SPLINE
SPL {X  -165.650, Y  +484.445, Z    +0.000, E1   +32.277, E3 +451169.154}
SPL {X  -165.650, Y  +481.524, Z    +0.000, E1   +31.089, E3 +451186.605}
SPL {X  -165.650, Y  +478.014, Z    +0.000, E1   +30.826, E3 +451200.213}
SPL {X  -165.650, Y  +474.473, Z    +0.000, E1   +30.943, E3 +451211.537}
SPL {X  -165.650, Y  +470.376, Z    +0.000, E1   +30.888, E3 +451226.066}
SPL {X  -165.650, Y  +465.146, Z    +0.000, E1   +30.883, E3 +451243.997}
SPL {X  -165.650, Y  +461.106, Z    +0.000, E1   +30.916, E3 +451257.415}
SPL {X  -165.650, Y  +458.435, Z    +0.000, E1   +30.759, E3 +451267.623}
SPL {X  -165.650, Y  +454.220, Z    +0.000, E1   +30.954, E3 +451280.856}
SPL {X  -165.650, Y  +450.433, Z    +0.000, E1   +30.789, E3 +451294.821}
SPL {X  -165.650, Y  +447.097, Z    +0.000, E1   +30.843, E3 +451305.869}
SPL {X  -165.650, Y  +443.673, Z    +0.000, E1   +30.907, E3 +451317.177}
SPL {X  -165.650, Y  +440.976, Z    +0.000, E1   +30.719, E3 +451327.633}
SPL {X  -165.650, Y  +436.324, Z    +0.000, E1   +30.994, E3 +451341.920}
SPL {X  -165.650, Y  +432.765, Z    +0.000, E1   +30.831, E3 +451354.920}
SPL {X  -165.650, Y  +429.309, Z    +0.000, E1   +30.920, E3 +451366.261}
SPL {X  -165.650, Y  +424.918, Z    +0.000, E1   +30.862, E3 +451381.718}
SPL {X  -165.650, Y  +421.437, Z    +0.000, E1   +30.833, E3 +451393.686}
SPL {X  -165.650, Y  +418.489, Z    +0.000, E1   +30.835, E3 +451403.803}
SPL {X  -165.650, Y  +415.831, Z    +0.000, E1   +30.847, E3 +451412.765}
SPL {X  -165.650, Y  +412.139, Z    +0.000, E1   +30.870, E3 +451425.476}
SPL {X  -165.650, Y  +406.834, Z    +0.000, E1   +30.919, E3 +451443.305}
SPL {X  -165.650, Y  +402.516, Z    +0.000, E1   +30.874, E3 +451458.227}
SPL {X  -165.650, Y  +398.147, Z    +0.000, E1   +30.902, E3 +451473.105}
SPL {X  -165.650, Y  +394.694, Z    +0.000, E1   +30.805, E3 +451485.414}
SPL {X  -165.650, Y  +391.522, Z    +0.000, E1   +30.837, E3 +451496.095}
SPL {X  -165.650, Y  +387.533, Z    +0.000, E1   +30.858, E3 +451509.721}
SPL {X  -165.650, Y  +383.627, Z    +0.000, E1   +30.885, E3 +451522.781}
SPL {X  -165.650, Y  +380.752, Z    +0.000, E1   +30.927, E3 +451532.295}
SPL {X  -165.648, Y  +377.739, Z    +0.000, E1   +30.835, E3 +451543.304}
SPL {X  -165.594, Y  +374.183, Z    +0.000, E1   +30.878, E3 +451555.141}
SPL {X  -165.492, Y  +371.263, Z    +0.000, E1   +30.913, E3 +451564.836}
SPL {X  -165.379, Y  +369.027, Z    +0.000, E1   +30.727, E3 +451573.775}
SPL {X  -165.167, Y  +365.866, Z    +0.000, E1   +30.741, E3 +451584.549}
SPL {X  -164.892, Y  +362.671, Z    +0.000, E1   +30.830, E3 +451594.873}
SPL {X  -164.570, Y  +359.612, Z    +0.000, E1   +30.773, E3 +451605.686}
SPL {X  -164.104, Y  +355.923, Z    +0.000, E1   +30.626, E3 +451619.402}
SPL {X  -163.573, Y  +352.353, Z    +0.000, E1   +30.451, E3 +451632.667}
SPL {X  -162.976, Y  +348.856, Z    +0.000, E1   +30.757, E3 +451642.591}
SPL {X  -161.497, Y  +341.640, Z    +0.000, E1   +33.276, E3 +451649.868}
SPL {X  -152.976, Y  +314.952, Z    +0.000, E1   +38.607, E3 +451694.213}
SPL {X  -137.967, Y  +286.821, Z    +0.000, E1   +43.969, E3 +451737.434}
ENDSPLINE

SPLINE
SPL {X  -153.316, Y  +315.777, Z    +0.000, E1   +33.140, E3 +451780.061}
SPL {X  -164.446, Y  +358.564, Z    +0.000, E1   +15.149, E3 +451745.272}
SPL {X  -165.510, Y  +371.680, Z    +0.000, E1    +7.684, E3 +451749.328}
SPL {X  -165.628, Y  +375.818, Z    +0.000, E1    +5.016, E3 +451757.257}
SPL {X  -165.650, Y  +383.362, Z    +0.000, E1    +0.177, E3 +451738.291}
SPL {X  -165.650, Y  +383.923, Z    +0.000, E1    -0.215, E3 +451751.448}
SPL {X  -165.650, Y  +388.083, Z    +0.000, E1    -3.355, E3 +451750.312}
SPL {X  -165.650, Y  +393.983, Z    +0.000, E1    -8.501, E3 +451746.710}
SPL {X  -165.650, Y  +402.241, Z    +0.000, E1   -16.711, E3 +451741.222}
SPL {X  -165.650, Y  +414.811, Z    +0.000, E1   -28.314, E3 +451740.752}
SPL {X  -165.650, Y  +423.479, Z    +0.000, E1   -29.012, E3 +451764.681}
SPL {X  -165.650, Y  +441.276, Z    +0.000, E1   -37.343, E3 +451776.370}
SPL {X  -165.650, Y  +462.890, Z    +0.000, E1   -40.484, E3 +451810.453}
ENDSPLINE

SPLINE
SPL {X  -165.650, Y  +446.920, Z    +0.000, E1   -31.238, E3 +451822.779}
ENDSPLINE

SPLINE
SPL {X  -165.650, Y  +447.935, Z    +0.000, E1   -30.213, E3 +451833.067}
SPL {X  -165.650, Y  +451.020, Z    +0.000, E1   -30.224, E3 +451843.887}
SPL {X  -165.650, Y  +454.519, Z    +0.000, E1   -30.374, E3 +451855.069}
SPL {X  -165.650, Y  +457.429, Z    +0.000, E1   -30.029, E3 +451867.771}
SPL {X  -165.650, Y  +461.678, Z    +0.000, E1   -30.426, E3 +451879.896}
SPL {X  -165.650, Y  +463.853, Z    +0.000, E1   -30.103, E3 +451889.735}
SPL {X  -165.650, Y  +468.397, Z    +0.000, E1   -30.302, E3 +451904.539}
SPL {X  -165.650, Y  +472.566, Z    +0.000, E1   -30.124, E3 +451920.248}
SPL {X  -165.650, Y  +476.540, Z    +0.000, E1   -30.193, E3 +451933.792}
SPL {X  -165.650, Y  +481.042, Z    +0.000, E1   -30.192, E3 +451949.738}
SPL {X  -165.650, Y  +485.236, Z    +0.000, E1   -30.294, E3 +451963.593}
SPL {X  -165.650, Y  +489.057, Z    +0.000, E1   -30.341, E3 +451976.799}
SPL {X  -165.650, Y  +491.647, Z    +0.000, E1   -29.894, E3 +451988.733}
SPL {X  -165.650, Y  +495.051, Z    +0.000, E1   -30.213, E3 +451998.661}
SPL {X  -165.650, Y  +498.418, Z    +0.000, E1   -30.282, E3 +452009.954}
SPL {X  -165.650, Y  +502.421, Z    +0.000, E1   -30.263, E3 +452024.312}
SPL {X  -165.650, Y  +506.344, Z    +0.000, E1   -30.129, E3 +452038.841}
SPL {X  -165.650, Y  +509.866, Z    +0.000, E1   -30.236, E3 +452050.511}
SPL {X  -165.650, Y  +513.685, Z    +0.000, E1   -30.234, E3 +452064.007}
SPL {X  -165.650, Y  +517.104, Z    +0.000, E1   -30.280, E3 +452075.559}
SPL {X  -165.650, Y  +520.621, Z    +0.000, E1   -30.198, E3 +452088.638}
SPL {X  -165.650, Y  +525.344, Z    +0.000, E1   -30.269, E3 +452104.695}
SPL {X  -165.650, Y  +528.152, Z    +0.000, E1   -29.991, E3 +452116.336}
SPL {X  -165.650, Y  +531.783, Z    +0.000, E1   -30.416, E3 +452126.229}
SPL {X  -165.650, Y  +534.115, Z    +0.000, E1   -30.089, E3 +452136.611}
SPL {X  -165.650, Y  +537.522, Z    +0.000, E1   -30.251, E3 +452147.525}
SPL {X  -165.650, Y  +540.621, Z    +0.000, E1   -30.014, E3 +452160.086}
SPL {X  -165.650, Y  +544.944, Z    +0.000, E1   -30.447, E3 +452172.286}
SPL {X  -165.650, Y  +547.199, Z    +0.000, E1   -30.132, E3 +452182.259}
SPL {X  -165.650, Y  +550.512, Z    +0.000, E1   -30.197, E3 +452193.585}
SPL {X  -165.650, Y  +553.852, Z    +0.000, E1   -30.156, E3 +452205.526}
SPL {X  -165.650, Y  +557.277, Z    +0.000, E1   -30.150, E3 +452217.700}
SPL {X  -165.650, Y  +561.168, Z    +0.000, E1   -30.194, E3 +452231.082}
SPL {X  -165.650, Y  +565.528, Z    +0.000, E1   -30.192, E3 +452246.564}
SPL {X  -165.650, Y  +570.048, Z    +0.000, E1   -30.238, E3 +452261.996}
SPL {X  -165.650, Y  +573.110, Z    +0.000, E1   -30.057, E3 +452273.981}
SPL {X  -165.650, Y  +577.587, Z    +0.000, E1   -30.270, E3 +452288.419}
SPL {X  -165.650, Y  +581.190, Z    +0.000, E1   -30.107, E3 +452302.059}
SPL {X  -165.650, Y  +585.053, Z    +0.000, E1   -30.090, E3 +452315.929}
ENDSPLINE

SPLINE
SPL {X  -165.650, Y  +484.445, Z    +0.000, E1   +32.277, E3 +452333.334}
SPL {X  -165.650, Y  +481.524, Z    +0.000, E1   +31.089, E3 +452350.784}
SPL {X  -165.650, Y  +478.014, Z    +0.000, E1   +30.826, E3 +452364.392}
SPL {X  -165.650, Y  +474.473, Z    +0.000, E1   +30.943, E3 +452375.716}
SPL {X  -165.650, Y  +470.376, Z    +0.000, E1   +30.888, E3 +452390.246}
SPL {X  -165.650, Y  +465.146, Z    +0.000, E1   +30.883, E3 +452408.176}
SPL {X  -165.650, Y  +461.106, Z    +0.000, E1   +30.916, E3 +452421.594}
SPL {X  -165.650, Y  +458.435, Z    +0.000, E1   +30.759, E3 +452431.802}
SPL {X  -165.650, Y  +454.220, Z    +0.000, E1   +30.954, E3 +452445.035}
SPL {X  -165.650, Y  +450.433, Z    +0.000, E1   +30.789, E3 +452459.000}
SPL {X  -165.650, Y  +447.097, Z    +0.000, E1   +30.843, E3 +452470.048}
SPL {X  -165.650, Y  +443.673, Z    +0.000, E1   +30.907, E3 +452481.356}
SPL {X  -165.650, Y  +440.976, Z    +0.000, E1   +30.719, E3 +452491.812}
SPL {X  -165.650, Y  +436.324, Z    +0.000, E1   +30.994, E3 +452506.099}
SPL {X  -165.650, Y  +432.765, Z    +0.000, E1   +30.831, E3 +452519.099}
SPL {X  -165.650, Y  +429.309, Z    +0.000, E1   +30.920, E3 +452530.440}
SPL {X  -165.650, Y  +424.918, Z    +0.000, E1   +30.862, E3 +452545.897}
SPL {X  -165.650, Y  +421.437, Z    +0.000, E1   +30.833, E3 +452557.865}
SPL {X  -165.650, Y  +417.366, Z    +0.000, E1   +30.879, E3 +452571.706}
SPL {X  -165.650, Y  +412.139, Z    +0.000, E1   +30.870, E3 +452589.655}
SPL {X  -165.650, Y  +406.834, Z    +0.000, E1   +30.919, E3 +452607.484}
SPL {X  -165.650, Y  +402.516, Z    +0.000, E1   +30.874, E3 +452622.406}
SPL {X  -165.650, Y  +398.147, Z    +0.000, E1   +30.902, E3 +452637.285}
SPL {X  -165.650, Y  +394.694, Z    +0.000, E1   +30.805, E3 +452649.593}
SPL {X  -165.650, Y  +391.522, Z    +0.000, E1   +30.837, E3 +452660.274}
SPL {X  -165.650, Y  +387.533, Z    +0.000, E1   +30.858, E3 +452673.900}
SPL {X  -165.650, Y  +383.627, Z    +0.000, E1   +30.885, E3 +452686.960}
SPL {X  -165.650, Y  +380.752, Z    +0.000, E1   +30.927, E3 +452696.474}
SPL {X  -165.648, Y  +377.739, Z    +0.000, E1   +30.835, E3 +452707.484}
SPL {X  -165.594, Y  +374.183, Z    +0.000, E1   +30.878, E3 +452719.320}
SPL {X  -165.492, Y  +371.263, Z    +0.000, E1   +30.913, E3 +452729.015}
SPL {X  -165.379, Y  +369.027, Z    +0.000, E1   +30.727, E3 +452737.954}
SPL {X  -165.167, Y  +365.866, Z    +0.000, E1   +30.741, E3 +452748.728}
SPL {X  -164.892, Y  +362.671, Z    +0.000, E1   +30.830, E3 +452759.052}
SPL {X  -164.570, Y  +359.612, Z    +0.000, E1   +30.773, E3 +452769.865}
SPL {X  -164.104, Y  +355.923, Z    +0.000, E1   +30.626, E3 +452783.581}
SPL {X  -163.573, Y  +352.353, Z    +0.000, E1   +30.451, E3 +452796.846}
SPL {X  -162.976, Y  +348.856, Z    +0.000, E1   +30.757, E3 +452806.770}
SPL {X  -161.497, Y  +341.640, Z    +0.000, E1   +33.276, E3 +452814.047}
SPL {X  -152.976, Y  +314.952, Z    +0.000, E1   +38.607, E3 +452858.392}
SPL {X  -137.967, Y  +286.821, Z    +0.000, E1   +43.969, E3 +452901.613}
ENDSPLINE

SPLINE
SPL {X  -149.143, Y  +306.414, Z    +0.000, E1   +36.361, E3 +452952.745}
SPL {X  -164.268, Y  +357.145, Z    +0.000, E1   +15.880, E3 +452910.505}
SPL {X  -165.510, Y  +371.680, Z    +0.000, E1    +7.684, E3 +452913.507}
SPL {X  -165.628, Y  +375.818, Z    +0.000, E1    +5.016, E3 +452921.436}
SPL {X  -165.650, Y  +383.362, Z    +0.000, E1    +0.177, E3 +452902.470}
SPL {X  -165.650, Y  +383.923, Z    +0.000, E1    -0.215, E3 +452915.627}
SPL {X  -165.650, Y  +388.083, Z    +0.000, E1    -3.355, E3 +452914.491}
SPL {X  -165.650, Y  +395.510, Z    +0.000, E1    -9.810, E3 +452910.617}
SPL {X  -165.650, Y  +403.066, Z    +0.000, E1   -17.886, E3 +452903.450}
SPL {X  -165.650, Y  +416.345, Z    +0.000, E1   -29.511, E3 +452905.193}
SPL {X  -165.650, Y  +422.331, Z    +0.000, E1   -27.760, E3 +452930.692}
SPL {X  -165.650, Y  +441.276, Z    +0.000, E1   -37.343, E3 +452940.549}
SPL {X  -165.650, Y  +462.890, Z    +0.000, E1   -40.484, E3 +452974.632}
ENDSPLINE

SPLINE
SPL {X  -165.650, Y  +446.920, Z    +0.000, E1   -31.238, E3 +452986.958}
ENDSPLINE

SPLINE
SPL {X  -165.650, Y  +447.935, Z    +0.000, E1   -30.213, E3 +452997.246}
SPL {X  -165.650, Y  +451.020, Z    +0.000, E1   -30.224, E3 +453008.066}
SPL {X  -165.650, Y  +454.519, Z    +0.000, E1   -30.374, E3 +453019.248}
SPL {X  -165.650, Y  +457.429, Z    +0.000, E1   -30.029, E3 +453031.950}
SPL {X  -165.650, Y  +461.678, Z    +0.000, E1   -30.426, E3 +453044.075}
SPL {X  -165.650, Y  +463.853, Z    +0.000, E1   -30.103, E3 +453053.914}
SPL {X  -165.650, Y  +468.397, Z    +0.000, E1   -30.302, E3 +453068.718}
SPL {X  -165.650, Y  +472.566, Z    +0.000, E1   -30.124, E3 +453084.428}
SPL {X  -165.650, Y  +476.540, Z    +0.000, E1   -30.193, E3 +453097.972}
SPL {X  -165.650, Y  +481.042, Z    +0.000, E1   -30.192, E3 +453113.917}
SPL {X  -165.650, Y  +485.236, Z    +0.000, E1   -30.294, E3 +453127.772}
SPL {X  -165.650, Y  +489.057, Z    +0.000, E1   -30.341, E3 +453140.978}
SPL {X  -165.650, Y  +491.647, Z    +0.000, E1   -29.894, E3 +453152.912}
SPL {X  -165.650, Y  +495.051, Z    +0.000, E1   -30.213, E3 +453162.841}
SPL {X  -165.650, Y  +499.546, Z    +0.000, E1   -30.283, E3 +453178.283}
SPL {X  -165.650, Y  +503.544, Z    +0.000, E1   -30.247, E3 +453192.352}
SPL {X  -165.650, Y  +506.344, Z    +0.000, E1   -30.129, E3 +453203.020}
SPL {X  -165.650, Y  +510.660, Z    +0.000, E1   -30.223, E3 +453217.724}
SPL {X  -165.650, Y  +514.670, Z    +0.000, E1   -30.278, E3 +453231.234}
SPL {X  -165.650, Y  +517.919, Z    +0.000, E1   -30.227, E3 +453243.093}
SPL {X  -165.650, Y  +522.822, Z    +0.000, E1   -30.289, E3 +453259.982}
SPL {X  -165.650, Y  +527.393, Z    +0.000, E1   -30.104, E3 +453277.230}
SPL {X  -165.650, Y  +531.783, Z    +0.000, E1   -30.416, E3 +453290.408}
SPL {X  -165.650, Y  +534.115, Z    +0.000, E1   -30.089, E3 +453300.790}
SPL {X  -165.650, Y  +537.522, Z    +0.000, E1   -30.251, E3 +453311.704}
SPL {X  -165.650, Y  +540.621, Z    +0.000, E1   -30.014, E3 +453324.265}
SPL {X  -165.650, Y  +544.944, Z    +0.000, E1   -30.447, E3 +453336.465}
SPL {X  -165.650, Y  +547.199, Z    +0.000, E1   -30.132, E3 +453346.438}
SPL {X  -165.650, Y  +550.512, Z    +0.000, E1   -30.197, E3 +453357.764}
SPL {X  -165.650, Y  +553.852, Z    +0.000, E1   -30.156, E3 +453369.705}
SPL {X  -165.650, Y  +557.277, Z    +0.000, E1   -30.150, E3 +453381.879}
SPL {X  -165.650, Y  +561.168, Z    +0.000, E1   -30.194, E3 +453395.261}
SPL {X  -165.650, Y  +564.449, Z    +0.000, E1   -30.167, E3 +453406.944}
SPL {X  -165.650, Y  +566.935, Z    +0.000, E1   -30.135, E3 +453415.850}
SPL {X  -165.650, Y  +570.048, Z    +0.000, E1   -30.238, E3 +453426.175}
SPL {X  -165.650, Y  +573.110, Z    +0.000, E1   -30.057, E3 +453438.160}
SPL {X  -165.650, Y  +576.497, Z    +0.000, E1   -30.234, E3 +453448.857}
SPL {X  -165.650, Y  +580.354, Z    +0.000, E1   -30.196, E3 +453462.873}
SPL {X  -165.650, Y  +585.053, Z    +0.000, E1   -30.090, E3 +453480.108}
ENDSPLINE

SPLINE
SPL {X  -165.650, Y  +484.445, Z    +0.000, E1   +32.277, E3 +453497.513}
SPL {X  -165.650, Y  +481.524, Z    +0.000, E1   +31.089, E3 +453514.963}
SPL {X  -165.650, Y  +478.014, Z    +0.000, E1   +30.826, E3 +453528.571}
SPL {X  -165.650, Y  +474.473, Z    +0.000, E1   +30.943, E3 +453539.895}
SPL {X  -165.650, Y  +471.826, Z    +0.000, E1   +30.770, E3 +453550.079}
SPL {X  -165.650, Y  +467.753, Z    +0.000, E1   +30.878, E3 +453563.452}
SPL {X  -165.650, Y  +463.837, Z    +0.000, E1   +30.924, E3 +453576.386}
SPL {X  -165.650, Y  +461.106, Z    +0.000, E1   +30.916, E3 +453585.773}
SPL {X  -165.650, Y  +458.435, Z    +0.000, E1   +30.759, E3 +453595.981}
SPL {X  -165.650, Y  +454.220, Z    +0.000, E1   +30.954, E3 +453609.214}
SPL {X  -165.650, Y  +450.433, Z    +0.000, E1   +30.789, E3 +453623.179}
SPL {X  -165.650, Y  +447.097, Z    +0.000, E1   +30.843, E3 +453634.227}
SPL {X  -165.650, Y  +443.673, Z    +0.000, E1   +30.907, E3 +453645.535}
SPL {X  -165.650, Y  +440.976, Z    +0.000, E1   +30.719, E3 +453655.992}
SPL {X  -165.650, Y  +436.324, Z    +0.000, E1   +30.994, E3 +453670.278}
SPL {X  -165.650, Y  +432.765, Z    +0.000, E1   +30.831, E3 +453683.278}
SPL {X  -165.650, Y  +429.309, Z    +0.000, E1   +30.920, E3 +453694.619}
SPL {X  -165.650, Y  +424.918, Z    +0.000, E1   +30.862, E3 +453710.076}
SPL {X  -165.650, Y  +421.437, Z    +0.000, E1   +30.833, E3 +453722.044}
SPL {X  -165.650, Y  +418.489, Z    +0.000, E1   +30.835, E3 +453732.161}
SPL {X  -165.650, Y  +414.127, Z    +0.000, E1   +30.869, E3 +453747.070}
SPL {X  -165.650, Y  +408.547, Z    +0.000, E1   +30.964, E3 +453765.485}
SPL {X  -165.650, Y  +405.433, Z    +0.000, E1   +30.730, E3 +453777.462}
SPL {X  -165.650, Y  +401.473, Z    +0.000, E1   +30.933, E3 +453789.911}
SPL {X  -165.650, Y  +396.018, Z    +0.000, E1   +30.861, E3 +453809.096}
SPL {X  -165.650, Y  +391.522, Z    +0.000, E1   +30.837, E3 +453824.453}
SPL {X  -165.650, Y  +387.533, Z    +0.000, E1   +30.858, E3 +453838.079}
SPL {X  -165.650, Y  +383.627, Z    +0.000, E1   +30.885, E3 +453851.139}
SPL {X  -165.650, Y  +380.752, Z    +0.000, E1   +30.927, E3 +453860.653}
SPL {X  -165.648, Y  +377.739, Z    +0.000, E1   +30.835, E3 +453871.663}
SPL {X  -165.594, Y  +374.183, Z    +0.000, E1   +30.878, E3 +453883.499}
SPL {X  -165.429, Y  +369.945, Z    +0.000, E1   +30.850, E3 +453898.375}
SPL {X  -165.167, Y  +365.866, Z    +0.000, E1   +30.741, E3 +453912.907}
SPL {X  -164.892, Y  +362.671, Z    +0.000, E1   +30.830, E3 +453923.231}
SPL {X  -164.570, Y  +359.612, Z    +0.000, E1   +30.773, E3 +453934.044}
SPL {X  -164.104, Y  +355.923, Z    +0.000, E1   +30.626, E3 +453947.760}
SPL {X  -163.573, Y  +352.353, Z    +0.000, E1   +30.451, E3 +453961.025}
SPL {X  -162.976, Y  +348.856, Z    +0.000, E1   +30.757, E3 +453970.949}
SPL {X  -161.497, Y  +341.640, Z    +0.000, E1   +33.276, E3 +453978.226}
SPL {X  -152.976, Y  +314.952, Z    +0.000, E1   +38.607, E3 +454022.571}
SPL {X  -137.967, Y  +286.821, Z    +0.000, E1   +43.969, E3 +454065.792}
ENDSPLINE

SPLINE
SPL {X  -149.143, Y  +306.414, Z    +0.000, E1   +36.361, E3 +454116.925}
SPL {X  -164.268, Y  +357.145, Z    +0.000, E1   +15.880, E3 +454074.684}
SPL {X  -165.510, Y  +371.680, Z    +0.000, E1    +7.684, E3 +454077.686}
SPL {X  -165.628, Y  +375.818, Z    +0.000, E1    +5.016, E3 +454085.615}
SPL {X  -165.650, Y  +383.362, Z    +0.000, E1    +0.177, E3 +454066.649}
SPL {X  -165.650, Y  +383.923, Z    +0.000, E1    -0.215, E3 +454079.807}
SPL {X  -165.650, Y  +388.083, Z    +0.000, E1    -3.355, E3 +454078.670}
SPL {X  -165.650, Y  +395.510, Z    +0.000, E1    -9.810, E3 +454074.796}
SPL {X  -165.650, Y  +403.066, Z    +0.000, E1   -17.886, E3 +454067.629}
SPL {X  -165.650, Y  +416.345, Z    +0.000, E1   -29.511, E3 +454069.372}
SPL {X  -165.650, Y  +422.331, Z    +0.000, E1   -27.760, E3 +454094.871}
SPL {X  -165.650, Y  +441.276, Z    +0.000, E1   -37.343, E3 +454104.728}
SPL {X  -165.650, Y  +462.890, Z    +0.000, E1   -40.484, E3 +454138.811}
ENDSPLINE

SPLINE
SPL {X  -165.650, Y  +446.920, Z    +0.000, E1   -31.238, E3 +454151.137}
ENDSPLINE

SPLINE
SPL {X  -165.650, Y  +447.935, Z    +0.000, E1   -30.213, E3 +454161.425}
SPL {X  -165.650, Y  +451.020, Z    +0.000, E1   -30.224, E3 +454172.245}
SPL {X  -165.650, Y  +454.519, Z    +0.000, E1   -30.374, E3 +454183.427}
SPL {X  -165.650, Y  +457.429, Z    +0.000, E1   -30.029, E3 +454196.129}
SPL {X  -165.650, Y  +461.678, Z    +0.000, E1   -30.426, E3 +454208.254}
SPL {X  -165.650, Y  +463.853, Z    +0.000, E1   -30.103, E3 +454218.093}
SPL {X  -165.650, Y  +468.397, Z    +0.000, E1   -30.302, E3 +454232.897}
SPL {X  -165.650, Y  +472.566, Z    +0.000, E1   -30.124, E3 +454248.607}
SPL {X  -165.650, Y  +475.265, Z    +0.000, E1   -30.034, E3 +454258.644}
SPL {X  -165.650, Y  +477.862, Z    +0.000, E1   -30.319, E3 +454265.836}
SPL {X  -165.650, Y  +481.042, Z    +0.000, E1   -30.192, E3 +454278.096}
SPL {X  -165.650, Y  +485.236, Z    +0.000, E1   -30.294, E3 +454291.951}
SPL {X  -165.650, Y  +488.041, Z    +0.000, E1   -30.253, E3 +454302.073}
SPL {X  -165.650, Y  +491.281, Z    +0.000, E1   -30.148, E3 +454314.211}
SPL {X  -165.650, Y  +495.051, Z    +0.000, E1   -30.213, E3 +454327.020}
SPL {X  -165.650, Y  +499.546, Z    +0.000, E1   -30.283, E3 +454342.462}
SPL {X  -165.650, Y  +503.544, Z    +0.000, E1   -30.247, E3 +454356.531}
SPL {X  -165.650, Y  +506.344, Z    +0.000, E1   -30.129, E3 +454367.200}
SPL {X  -165.650, Y  +510.660, Z    +0.000, E1   -30.223, E3 +454381.903}
SPL {X  -165.650, Y  +514.670, Z    +0.000, E1   -30.278, E3 +454395.413}
SPL {X  -165.650, Y  +517.919, Z    +0.000, E1   -30.227, E3 +454407.272}
SPL {X  -165.650, Y  +522.822, Z    +0.000, E1   -30.289, E3 +454424.161}
SPL {X  -165.650, Y  +527.393, Z    +0.000, E1   -30.104, E3 +454441.410}
SPL {X  -165.650, Y  +531.783, Z    +0.000, E1   -30.416, E3 +454454.587}
SPL {X  -165.650, Y  +534.115, Z    +0.000, E1   -30.089, E3 +454464.969}
SPL {X  -165.650, Y  +537.522, Z    +0.000, E1   -30.251, E3 +454475.883}
SPL {X  -165.650, Y  +540.621, Z    +0.000, E1   -30.014, E3 +454488.444}
SPL {X  -165.650, Y  +544.944, Z    +0.000, E1   -30.447, E3 +454500.644}
SPL {X  -165.650, Y  +547.199, Z    +0.000, E1   -30.132, E3 +454510.617}
SPL {X  -165.650, Y  +550.512, Z    +0.000, E1   -30.197, E3 +454521.943}
SPL {X  -165.650, Y  +553.852, Z    +0.000, E1   -30.156, E3 +454533.884}
SPL {X  -165.650, Y  +557.277, Z    +0.000, E1   -30.150, E3 +454546.058}
SPL {X  -165.650, Y  +561.168, Z    +0.000, E1   -30.194, E3 +454559.440}
SPL {X  -165.650, Y  +565.528, Z    +0.000, E1   -30.192, E3 +454574.923}
SPL {X  -165.650, Y  +570.048, Z    +0.000, E1   -30.238, E3 +454590.354}
SPL {X  -165.650, Y  +573.110, Z    +0.000, E1   -30.057, E3 +454602.339}
SPL {X  -165.650, Y  +577.587, Z    +0.000, E1   -30.270, E3 +454616.778}
SPL {X  -165.650, Y  +581.190, Z    +0.000, E1   -30.107, E3 +454630.417}
SPL {X  -165.650, Y  +585.053, Z    +0.000, E1   -30.090, E3 +454644.287}
ENDSPLINE

SPLINE
SPL {X  -165.650, Y  +484.445, Z    +0.000, E1   +32.277, E3 +454661.692}
SPL {X  -165.650, Y  +481.524, Z    +0.000, E1   +31.089, E3 +454679.142}
SPL {X  -165.650, Y  +478.014, Z    +0.000, E1   +30.826, E3 +454692.750}
SPL {X  -165.650, Y  +474.473, Z    +0.000, E1   +30.943, E3 +454704.074}
SPL {X  -165.650, Y  +471.826, Z    +0.000, E1   +30.770, E3 +454714.258}
SPL {X  -165.650, Y  +467.753, Z    +0.000, E1   +30.878, E3 +454727.631}
SPL {X  -165.650, Y  +463.837, Z    +0.000, E1   +30.924, E3 +454740.565}
SPL {X  -165.650, Y  +461.106, Z    +0.000, E1   +30.916, E3 +454749.952}
SPL {X  -165.650, Y  +457.156, Z    +0.000, E1   +30.860, E3 +454764.029}
SPL {X  -165.650, Y  +453.156, Z    +0.000, E1   +30.934, E3 +454777.003}
SPL {X  -165.650, Y  +450.433, Z    +0.000, E1   +30.789, E3 +454787.358}
SPL {X  -165.650, Y  +447.097, Z    +0.000, E1   +30.843, E3 +454798.407}
SPL {X  -165.650, Y  +443.673, Z    +0.000, E1   +30.907, E3 +454809.714}
SPL {X  -165.650, Y  +439.486, Z    +0.000, E1   +30.857, E3 +454824.523}
SPL {X  -165.650, Y  +435.146, Z    +0.000, E1   +30.969, E3 +454838.443}
SPL {X  -165.650, Y  +431.607, Z    +0.000, E1   +30.889, E3 +454851.157}
SPL {X  -165.650, Y  +427.340, Z    +0.000, E1   +30.870, E3 +454865.869}
SPL {X  -165.650, Y  +423.901, Z    +0.000, E1   +30.858, E3 +454877.625}
SPL {X  -165.650, Y  +421.437, Z    +0.000, E1   +30.833, E3 +454886.223}
SPL {X  -165.650, Y  +418.489, Z    +0.000, E1   +30.835, E3 +454896.340}
SPL {X  -165.650, Y  +414.127, Z    +0.000, E1   +30.869, E3 +454911.249}
SPL {X  -165.650, Y  +408.547, Z    +0.000, E1   +30.964, E3 +454929.664}
SPL {X  -165.650, Y  +405.433, Z    +0.000, E1   +30.730, E3 +454941.642}
SPL {X  -165.650, Y  +401.473, Z    +0.000, E1   +30.933, E3 +454954.090}
SPL {X  -165.650, Y  +396.018, Z    +0.000, E1   +30.861, E3 +454973.275}
SPL {X  -165.650, Y  +390.331, Z    +0.000, E1   +30.892, E3 +454992.527}
SPL {X  -165.650, Y  +384.849, Z    +0.000, E1   +30.885, E3 +455011.331}
SPL {X  -165.650, Y  +380.752, Z    +0.000, E1   +30.927, E3 +455024.832}
SPL {X  -165.648, Y  +377.739, Z    +0.000, E1   +30.835, E3 +455035.842}
SPL {X  -165.594, Y  +374.183, Z    +0.000, E1   +30.878, E3 +455047.679}
SPL {X  -165.492, Y  +371.263, Z    +0.000, E1   +30.913, E3 +455057.374}
SPL {X  -165.379, Y  +369.027, Z    +0.000, E1   +30.727, E3 +455066.312}
SPL {X  -165.167, Y  +365.866, Z    +0.000, E1   +30.741, E3 +455077.086}
SPL {X  -164.892, Y  +362.671, Z    +0.000, E1   +30.830, E3 +455087.410}
SPL {X  -164.570, Y  +359.612, Z    +0.000, E1   +30.773, E3 +455098.223}
SPL {X  -164.104, Y  +355.923, Z    +0.000, E1   +30.626, E3 +455111.939}
SPL {X  -163.573, Y  +352.353, Z    +0.000, E1   +30.451, E3 +455125.204}
SPL {X  -162.476, Y  +346.230, Z    +0.000, E1   +31.677, E3 +455137.785}
SPL {X  -152.976, Y  +314.952, Z    +0.000, E1   +38.607, E3 +455186.750}
SPL {X  -137.967, Y  +286.821, Z    +0.000, E1   +43.969, E3 +455229.971}
ENDSPLINE

SPLINE
SPL {X  -149.143, Y  +306.414, Z    +0.000, E1   +36.361, E3 +455281.104}
SPL {X  -163.091, Y  +349.496, Z    +0.000, E1   +19.699, E3 +455237.887}
SPL {X  -165.027, Y  +364.142, Z    +0.000, E1   +12.054, E3 +455241.027}
SPL {X  -165.612, Y  +374.969, Z    +0.000, E1    +5.630, E3 +455246.210}
SPL {X  -165.650, Y  +383.362, Z    +0.000, E1    +0.177, E3 +455230.828}
SPL {X  -165.650, Y  +383.923, Z    +0.000, E1    -0.215, E3 +455243.986}
SPL {X  -165.650, Y  +388.083, Z    +0.000, E1    -3.355, E3 +455242.849}
SPL {X  -165.650, Y  +393.983, Z    +0.000, E1    -8.501, E3 +455239.247}
SPL {X  -165.650, Y  +402.241, Z    +0.000, E1   -16.711, E3 +455233.759}
SPL {X  -165.650, Y  +416.345, Z    +0.000, E1   -29.511, E3 +455233.551}
SPL {X  -165.650, Y  +422.331, Z    +0.000, E1   -27.760, E3 +455259.050}
SPL {X  -165.650, Y  +441.276, Z    +0.000, E1   -37.343, E3 +455268.907}
SPL {X  -165.650, Y  +462.890, Z    +0.000, E1   -40.484, E3 +455302.990}
ENDSPLINE

SPLINE
SPL {X  -165.650, Y  +446.920, Z    +0.000, E1   -31.238, E3 +455315.316}
ENDSPLINE

SPLINE
SPL {X  -165.650, Y  +447.935, Z    +0.000, E1   -30.213, E3 +455325.604}
SPL {X  -165.650, Y  +451.020, Z    +0.000, E1   -30.224, E3 +455336.424}
SPL {X  -165.650, Y  +454.519, Z    +0.000, E1   -30.374, E3 +455347.607}
SPL {X  -165.650, Y  +456.542, Z    +0.000, E1   -29.986, E3 +455357.351}
SPL {X  -165.650, Y  +460.618, Z    +0.000, E1   -30.298, E3 +455369.672}
SPL {X  -165.650, Y  +463.853, Z    +0.000, E1   -30.103, E3 +455382.273}
SPL {X  -165.650, Y  +468.397, Z    +0.000, E1   -30.302, E3 +455397.076}
SPL {X  -165.650, Y  +472.566, Z    +0.000, E1   -30.124, E3 +455412.786}
SPL {X  -165.650, Y  +475.265, Z    +0.000, E1   -30.034, E3 +455422.823}
SPL {X  -165.650, Y  +477.862, Z    +0.000, E1   -30.319, E3 +455430.015}
SPL {X  -165.650, Y  +481.042, Z    +0.000, E1   -30.192, E3 +455442.275}
SPL {X  -165.650, Y  +485.236, Z    +0.000, E1   -30.294, E3 +455456.131}
SPL {X  -165.650, Y  +488.041, Z    +0.000, E1   -30.253, E3 +455466.252}
SPL {X  -165.650, Y  +491.281, Z    +0.000, E1   -30.148, E3 +455478.390}
SPL {X  -165.650, Y  +495.051, Z    +0.000, E1   -30.213, E3 +455491.199}
SPL {X  -165.650, Y  +499.546, Z    +0.000, E1   -30.283, E3 +455506.642}
SPL {X  -165.650, Y  +503.544, Z    +0.000, E1   -30.247, E3 +455520.710}
SPL {X  -165.650, Y  +506.344, Z    +0.000, E1   -30.129, E3 +455531.379}
SPL {X  -165.650, Y  +510.660, Z    +0.000, E1   -30.223, E3 +455546.082}
SPL {X  -165.650, Y  +514.670, Z    +0.000, E1   -30.278, E3 +455559.592}
SPL {X  -165.650, Y  +517.919, Z    +0.000, E1   -30.227, E3 +455571.451}
SPL {X  -165.650, Y  +521.521, Z    +0.000, E1   -30.210, E3 +455584.126}
SPL {X  -165.650, Y  +525.344, Z    +0.000, E1   -30.269, E3 +455597.232}
SPL {X  -165.650, Y  +528.152, Z    +0.000, E1   -29.991, E3 +455608.873}
SPL {X  -165.650, Y  +531.783, Z    +0.000, E1   -30.416, E3 +455618.766}
SPL {X  -165.650, Y  +534.115, Z    +0.000, E1   -30.089, E3 +455629.148}
SPL {X  -165.650, Y  +537.522, Z    +0.000, E1   -30.251, E3 +455640.062}
SPL {X  -165.650, Y  +540.621, Z    +0.000, E1   -30.014, E3 +455652.623}
SPL {X  -165.650, Y  +544.944, Z    +0.000, E1   -30.447, E3 +455664.823}
SPL {X  -165.650, Y  +547.199, Z    +0.000, E1   -30.132, E3 +455674.796}
SPL {X  -165.650, Y  +550.512, Z    +0.000, E1   -30.197, E3 +455686.122}
SPL {X  -165.650, Y  +553.852, Z    +0.000, E1   -30.156, E3 +455698.063}
SPL {X  -165.650, Y  +557.277, Z    +0.000, E1   -30.150, E3 +455710.238}
SPL {X  -165.650, Y  +561.168, Z    +0.000, E1   -30.194, E3 +455723.619}
SPL {X  -165.650, Y  +565.528, Z    +0.000, E1   -30.192, E3 +455739.102}
SPL {X  -165.650, Y  +570.048, Z    +0.000, E1   -30.238, E3 +455754.533}
SPL {X  -165.650, Y  +573.110, Z    +0.000, E1   -30.057, E3 +455766.518}
SPL {X  -165.650, Y  +576.497, Z    +0.000, E1   -30.234, E3 +455777.216}
SPL {X  -165.650, Y  +580.354, Z    +0.000, E1   -30.196, E3 +455791.231}
SPL {X  -165.650, Y  +585.053, Z    +0.000, E1   -30.090, E3 +455808.466}
ENDSPLINE

SPLINE
SPL {X  -165.650, Y  +484.968, Z    +0.000, E1   +32.508, E3 +455822.432}
SPL {X  -165.650, Y  +482.280, Z    +0.000, E1   +31.680, E3 +455836.759}
SPL {X  -165.650, Y  +481.693, Z    +0.000, E1   +30.334, E3 +455847.468}
SPL {X  -165.650, Y  +478.014, Z    +0.000, E1   +30.826, E3 +455856.929}
SPL {X  -165.650, Y  +474.473, Z    +0.000, E1   +30.943, E3 +455868.253}
SPL {X  -165.650, Y  +471.826, Z    +0.000, E1   +30.770, E3 +455878.437}
SPL {X  -165.650, Y  +467.753, Z    +0.000, E1   +30.878, E3 +455891.810}
SPL {X  -165.650, Y  +463.837, Z    +0.000, E1   +30.924, E3 +455904.744}
SPL {X  -165.650, Y  +461.106, Z    +0.000, E1   +30.916, E3 +455914.131}
SPL {X  -165.650, Y  +458.435, Z    +0.000, E1   +30.759, E3 +455924.339}
SPL {X  -165.650, Y  +454.220, Z    +0.000, E1   +30.954, E3 +455937.572}
SPL {X  -165.650, Y  +450.433, Z    +0.000, E1   +30.789, E3 +455951.537}
SPL {X  -165.650, Y  +447.097, Z    +0.000, E1   +30.843, E3 +455962.586}
SPL {X  -165.650, Y  +443.673, Z    +0.000, E1   +30.907, E3 +455973.893}
SPL {X  -165.650, Y  +440.976, Z    +0.000, E1   +30.719, E3 +455984.350}
SPL {X  -165.650, Y  +437.973, Z    +0.000, E1   +30.928, E3 +455993.222}
SPL {X  -165.650, Y  +434.043, Z    +0.000, E1   +30.950, E3 +456006.719}
SPL {X  -165.650, Y  +430.419, Z    +0.000, E1   +30.895, E3 +456019.222}
SPL {X  -165.650, Y  +427.340, Z    +0.000, E1   +30.870, E3 +456030.048}
SPL {X  -165.650, Y  +422.641, Z    +0.000, E1   +30.884, E3 +456046.137}
SPL {X  -165.650, Y  +418.489, Z    +0.000, E1   +30.835, E3 +456060.519}
SPL {X  -165.650, Y  +414.127, Z    +0.000, E1   +30.869, E3 +456075.428}
SPL {X  -165.650, Y  +408.547, Z    +0.000, E1   +30.964, E3 +456093.843}
SPL {X  -165.650, Y  +405.433, Z    +0.000, E1   +30.730, E3 +456105.821}
SPL {X  -165.650, Y  +402.516, Z    +0.000, E1   +30.874, E3 +456114.943}
SPL {X  -165.650, Y  +398.147, Z    +0.000, E1   +30.902, E3 +456129.822}
SPL {X  -165.650, Y  +394.694, Z    +0.000, E1   +30.805, E3 +456142.130}
SPL {X  -165.650, Y  +391.522, Z    +0.000, E1   +30.837, E3 +456152.811}
SPL {X  -165.650, Y  +387.533, Z    +0.000, E1   +30.858, E3 +456166.437}
SPL {X  -165.650, Y  +383.627, Z    +0.000, E1   +30.885, E3 +456179.497}
SPL {X  -165.650, Y  +379.886, Z    +0.000, E1   +30.887, E3 +456192.386}
SPL {X  -165.614, Y  +375.058, Z    +0.000, E1   +30.905, E3 +456208.839}
SPL {X  -165.492, Y  +371.263, Z    +0.000, E1   +30.913, E3 +456221.553}
SPL {X  -165.379, Y  +369.027, Z    +0.000, E1   +30.727, E3 +456230.491}
SPL {X  -165.167, Y  +365.866, Z    +0.000, E1   +30.741, E3 +456241.265}
SPL {X  -164.892, Y  +362.671, Z    +0.000, E1   +30.830, E3 +456251.589}
SPL {X  -164.570, Y  +359.612, Z    +0.000, E1   +30.773, E3 +456262.402}
SPL {X  -164.104, Y  +355.923, Z    +0.000, E1   +30.626, E3 +456276.118}
SPL {X  -163.573, Y  +352.353, Z    +0.000, E1   +30.451, E3 +456289.383}
SPL {X  -162.976, Y  +348.856, Z    +0.000, E1   +30.757, E3 +456299.307}
SPL {X  -161.497, Y  +341.640, Z    +0.000, E1   +33.276, E3 +456306.585}
SPL {X  -152.976, Y  +314.952, Z    +0.000, E1   +38.607, E3 +456350.929}
SPL {X  -137.967, Y  +286.821, Z    +0.000, E1   +43.969, E3 +456394.150}
ENDSPLINE

SPLINE
SPL {X  -149.143, Y  +306.414, Z    +0.000, E1   +36.361, E3 +456445.283}
SPL {X  -164.268, Y  +357.145, Z    +0.000, E1   +15.880, E3 +456403.042}
SPL {X  -165.379, Y  +369.025, Z    +0.000, E1    +9.158, E3 +456407.713}
SPL {X  -165.612, Y  +374.969, Z    +0.000, E1    +5.630, E3 +456410.389}
SPL {X  -165.650, Y  +383.362, Z    +0.000, E1    +0.177, E3 +456395.007}
SPL {X  -165.650, Y  +383.923, Z    +0.000, E1    -0.215, E3 +456408.165}
SPL {X  -165.650, Y  +388.083, Z    +0.000, E1    -3.355, E3 +456407.028}
SPL {X  -165.650, Y  +393.983, Z    +0.000, E1    -8.501, E3 +456403.426}
SPL {X  -165.650, Y  +402.241, Z    +0.000, E1   -16.711, E3 +456397.938}
SPL {X  -165.650, Y  +416.345, Z    +0.000, E1   -29.511, E3 +456397.730}
SPL {X  -165.650, Y  +422.331, Z    +0.000, E1   -27.760, E3 +456423.229}
SPL {X  -165.650, Y  +441.276, Z    +0.000, E1   -37.343, E3 +456433.086}
SPL {X  -165.650, Y  +462.890, Z    +0.000, E1   -40.484, E3 +456467.169}
ENDSPLINE

SPLINE
SPL {X  -165.650, Y  +446.920, Z    +0.000, E1   -31.238, E3 +456479.495}
ENDSPLINE

SPLINE
SPL {X  -165.650, Y  +447.935, Z    +0.000, E1   -30.213, E3 +456489.783}
SPL {X  -165.650, Y  +451.020, Z    +0.000, E1   -30.224, E3 +456500.603}
SPL {X  -165.650, Y  +454.519, Z    +0.000, E1   -30.374, E3 +456511.786}
SPL {X  -165.650, Y  +456.542, Z    +0.000, E1   -29.986, E3 +456521.530}
SPL {X  -165.650, Y  +460.618, Z    +0.000, E1   -30.298, E3 +456533.851}
SPL {X  -165.650, Y  +463.853, Z    +0.000, E1   -30.103, E3 +456546.452}
SPL {X  -165.650, Y  +468.397, Z    +0.000, E1   -30.302, E3 +456561.256}
SPL {X  -165.650, Y  +472.566, Z    +0.000, E1   -30.124, E3 +456576.965}
SPL {X  -165.650, Y  +476.540, Z    +0.000, E1   -30.193, E3 +456590.509}
SPL {X  -165.650, Y  +480.320, Z    +0.000, E1   -30.163, E3 +456603.987}
SPL {X  -165.650, Y  +484.477, Z    +0.000, E1   -30.274, E3 +456617.876}
SPL {X  -165.650, Y  +488.041, Z    +0.000, E1   -30.253, E3 +456630.431}
SPL {X  -165.650, Y  +491.281, Z    +0.000, E1   -30.148, E3 +456642.569}
SPL {X  -165.650, Y  +495.051, Z    +0.000, E1   -30.213, E3 +456655.378}
SPL {X  -165.650, Y  +499.546, Z    +0.000, E1   -30.283, E3 +456670.821}
SPL {X  -165.650, Y  +503.544, Z    +0.000, E1   -30.247, E3 +456684.889}
SPL {X  -165.650, Y  +506.344, Z    +0.000, E1   -30.129, E3 +456695.558}
SPL {X  -165.650, Y  +509.866, Z    +0.000, E1   -30.236, E3 +456707.227}
SPL {X  -165.650, Y  +513.685, Z    +0.000, E1   -30.234, E3 +456720.723}
SPL {X  -165.650, Y  +517.919, Z    +0.000, E1   -30.227, E3 +456735.630}
SPL {X  -165.650, Y  +521.521, Z    +0.000, E1   -30.210, E3 +456748.305}
SPL {X  -165.650, Y  +525.344, Z    +0.000, E1   -30.269, E3 +456761.411}
SPL {X  -165.650, Y  +528.152, Z    +0.000, E1   -29.991, E3 +456773.052}
SPL {X  -165.650, Y  +531.783, Z    +0.000, E1   -30.416, E3 +456782.945}
SPL {X  -165.650, Y  +534.115, Z    +0.000, E1   -30.089, E3 +456793.327}
SPL {X  -165.650, Y  +537.522, Z    +0.000, E1   -30.251, E3 +456804.241}
SPL {X  -165.650, Y  +540.621, Z    +0.000, E1   -30.014, E3 +456816.802}
SPL {X  -165.650, Y  +544.944, Z    +0.000, E1   -30.447, E3 +456829.002}
SPL {X  -165.650, Y  +547.199, Z    +0.000, E1   -30.132, E3 +456838.976}
SPL {X  -165.650, Y  +550.512, Z    +0.000, E1   -30.197, E3 +456850.301}
SPL {X  -165.650, Y  +553.852, Z    +0.000, E1   -30.156, E3 +456862.242}
SPL {X  -165.650, Y  +557.277, Z    +0.000, E1   -30.150, E3 +456874.417}
SPL {X  -165.650, Y  +561.168, Z    +0.000, E1   -30.194, E3 +456887.798}
SPL {X  -165.650, Y  +565.528, Z    +0.000, E1   -30.192, E3 +456903.281}
SPL {X  -165.650, Y  +570.048, Z    +0.000, E1   -30.238, E3 +456918.712}
SPL {X  -165.650, Y  +573.110, Z    +0.000, E1   -30.057, E3 +456930.697}
SPL {X  -165.650, Y  +577.587, Z    +0.000, E1   -30.270, E3 +456945.136}
SPL {X  -165.650, Y  +581.190, Z    +0.000, E1   -30.107, E3 +456958.775}
SPL {X  -165.650, Y  +585.053, Z    +0.000, E1   -30.090, E3 +456972.645}
ENDSPLINE

SPLINE
SPL {X  -165.650, Y  +484.445, Z    +0.000, E1   +32.277, E3 +456990.050}
SPL {X  -165.650, Y  +481.524, Z    +0.000, E1   +31.089, E3 +457007.500}
SPL {X  -165.650, Y  +478.014, Z    +0.000, E1   +30.826, E3 +457021.108}
SPL {X  -165.650, Y  +474.473, Z    +0.000, E1   +30.943, E3 +457032.432}
SPL {X  -165.650, Y  +471.826, Z    +0.000, E1   +30.770, E3 +457042.616}
SPL {X  -165.650, Y  +467.753, Z    +0.000, E1   +30.878, E3 +457055.989}
SPL {X  -165.650, Y  +463.837, Z    +0.000, E1   +30.924, E3 +457068.923}
SPL {X  -165.650, Y  +461.106, Z    +0.000, E1   +30.916, E3 +457078.310}
SPL {X  -165.650, Y  +457.156, Z    +0.000, E1   +30.860, E3 +457092.387}
SPL {X  -165.650, Y  +453.156, Z    +0.000, E1   +30.934, E3 +457105.361}
SPL {X  -165.650, Y  +450.433, Z    +0.000, E1   +30.789, E3 +457115.716}
SPL {X  -165.650, Y  +447.097, Z    +0.000, E1   +30.843, E3 +457126.765}
SPL {X  -165.650, Y  +443.673, Z    +0.000, E1   +30.907, E3 +457138.072}
SPL {X  -165.650, Y  +439.486, Z    +0.000, E1   +30.857, E3 +457152.882}
SPL {X  -165.650, Y  +435.146, Z    +0.000, E1   +30.969, E3 +457166.801}
SPL {X  -165.650, Y  +432.765, Z    +0.000, E1   +30.831, E3 +457175.815}
SPL {X  -165.650, Y  +429.309, Z    +0.000, E1   +30.920, E3 +457187.156}
SPL {X  -165.650, Y  +424.918, Z    +0.000, E1   +30.862, E3 +457202.613}
SPL {X  -165.650, Y  +421.437, Z    +0.000, E1   +30.833, E3 +457214.582}
SPL {X  -165.650, Y  +417.366, Z    +0.000, E1   +30.879, E3 +457228.422}
SPL {X  -165.650, Y  +413.181, Z    +0.000, E1   +30.815, E3 +457243.020}
SPL {X  -165.650, Y  +408.547, Z    +0.000, E1   +30.964, E3 +457258.023}
SPL {X  -165.650, Y  +403.421, Z    +0.000, E1   +30.863, E3 +457276.240}
SPL {X  -165.650, Y  +399.681, Z    +0.000, E1   +30.933, E3 +457288.323}
SPL {X  -165.650, Y  +396.018, Z    +0.000, E1   +30.861, E3 +457301.633}
SPL {X  -165.650, Y  +391.522, Z    +0.000, E1   +30.837, E3 +457316.990}
SPL {X  -165.650, Y  +387.533, Z    +0.000, E1   +30.858, E3 +457330.616}
SPL {X  -165.650, Y  +383.627, Z    +0.000, E1   +30.885, E3 +457343.677}
SPL {X  -165.650, Y  +380.752, Z    +0.000, E1   +30.927, E3 +457353.190}
SPL {X  -165.648, Y  +377.739, Z    +0.000, E1   +30.835, E3 +457364.200}
SPL {X  -165.594, Y  +374.183, Z    +0.000, E1   +30.878, E3 +457376.037}
SPL {X  -165.429, Y  +369.945, Z    +0.000, E1   +30.850, E3 +457390.912}
SPL {X  -165.167, Y  +365.866, Z    +0.000, E1   +30.741, E3 +457405.444}
SPL {X  -164.892, Y  +362.671, Z    +0.000, E1   +30.830, E3 +457415.768}
SPL {X  -164.570, Y  +359.612, Z    +0.000, E1   +30.773, E3 +457426.581}
SPL {X  -164.104, Y  +355.923, Z    +0.000, E1   +30.626, E3 +457440.298}
SPL {X  -163.573, Y  +352.353, Z    +0.000, E1   +30.451, E3 +457453.562}
SPL {X  -162.476, Y  +346.230, Z    +0.000, E1   +31.677, E3 +457466.143}
SPL {X  -152.976, Y  +314.952, Z    +0.000, E1   +38.607, E3 +457515.108}
SPL {X  -137.967, Y  +286.821, Z    +0.000, E1   +43.969, E3 +457558.329}
ENDSPLINE

SPLINE
SPL {X  -153.316, Y  +315.777, Z    +0.000, E1   +33.140, E3 +457600.957}
SPL {X  -164.446, Y  +358.564, Z    +0.000, E1   +15.149, E3 +457566.168}
SPL {X  -165.510, Y  +371.680, Z    +0.000, E1    +7.684, E3 +457570.223}
SPL {X  -165.628, Y  +375.818, Z    +0.000, E1    +5.016, E3 +457578.153}
SPL {X  -165.650, Y  +383.362, Z    +0.000, E1    +0.177, E3 +457559.186}
SPL {X  -165.650, Y  +383.923, Z    +0.000, E1    -0.215, E3 +457572.344}
SPL {X  -165.650, Y  +388.083, Z    +0.000, E1    -3.355, E3 +457571.207}
SPL {X  -165.650, Y  +393.983, Z    +0.000, E1    -8.501, E3 +457567.606}
SPL {X  -165.650, Y  +402.241, Z    +0.000, E1   -16.711, E3 +457562.117}
SPL {X  -165.650, Y  +414.811, Z    +0.000, E1   -28.314, E3 +457561.648}
SPL {X  -165.650, Y  +423.479, Z    +0.000, E1   -29.012, E3 +457585.576}
SPL {X  -165.650, Y  +441.276, Z    +0.000, E1   -37.343, E3 +457597.265}
SPL {X  -165.650, Y  +462.890, Z    +0.000, E1   -40.484, E3 +457631.348}
ENDSPLINE

SPLINE
SPL {X  -165.650, Y  +446.920, Z    +0.000, E1   -31.238, E3 +457643.674}
ENDSPLINE

SPLINE
SPL {X  -165.650, Y  +447.935, Z    +0.000, E1   -30.213, E3 +457653.962}
SPL {X  -165.650, Y  +451.020, Z    +0.000, E1   -30.224, E3 +457664.782}
SPL {X  -165.650, Y  +454.519, Z    +0.000, E1   -30.374, E3 +457675.965}
SPL {X  -165.650, Y  +456.542, Z    +0.000, E1   -29.986, E3 +457685.709}
SPL {X  -165.650, Y  +460.618, Z    +0.000, E1   -30.298, E3 +457698.030}
SPL {X  -165.650, Y  +463.853, Z    +0.000, E1   -30.103, E3 +457710.631}
SPL {X  -165.650, Y  +468.397, Z    +0.000, E1   -30.302, E3 +457725.435}
SPL {X  -165.650, Y  +472.566, Z    +0.000, E1   -30.124, E3 +457741.144}
SPL {X  -165.650, Y  +476.540, Z    +0.000, E1   -30.193, E3 +457754.688}
SPL {X  -165.650, Y  +480.320, Z    +0.000, E1   -30.163, E3 +457768.166}
SPL {X  -165.650, Y  +484.477, Z    +0.000, E1   -30.274, E3 +457782.055}
SPL {X  -165.650, Y  +488.041, Z    +0.000, E1   -30.253, E3 +457794.610}
SPL {X  -165.650, Y  +491.281, Z    +0.000, E1   -30.148, E3 +457806.748}
SPL {X  -165.650, Y  +495.051, Z    +0.000, E1   -30.213, E3 +457819.557}
SPL {X  -165.650, Y  +498.418, Z    +0.000, E1   -30.282, E3 +457830.850}
SPL {X  -165.650, Y  +500.833, Z    +0.000, E1   -30.191, E3 +457839.899}
SPL {X  -165.650, Y  +504.246, Z    +0.000, E1   -30.231, E3 +457851.765}
SPL {X  -165.650, Y  +507.017, Z    +0.000, E1   -30.108, E3 +457862.174}
SPL {X  -165.650, Y  +510.660, Z    +0.000, E1   -30.223, E3 +457874.440}
SPL {X  -165.650, Y  +514.670, Z    +0.000, E1   -30.278, E3 +457887.950}
SPL {X  -165.650, Y  +517.919, Z    +0.000, E1   -30.227, E3 +457899.810}
SPL {X  -165.650, Y  +522.822, Z    +0.000, E1   -30.289, E3 +457916.699}
SPL {X  -165.650, Y  +527.393, Z    +0.000, E1   -30.104, E3 +457933.947}
SPL {X  -165.650, Y  +531.783, Z    +0.000, E1   -30.416, E3 +457947.124}
SPL {X  -165.650, Y  +534.115, Z    +0.000, E1   -30.089, E3 +457957.506}
SPL {X  -165.650, Y  +537.522, Z    +0.000, E1   -30.251, E3 +457968.421}
SPL {X  -165.650, Y  +540.621, Z    +0.000, E1   -30.014, E3 +457980.982}
SPL {X  -165.650, Y  +544.944, Z    +0.000, E1   -30.447, E3 +457993.181}
SPL {X  -165.650, Y  +548.549, Z    +0.000, E1   -30.216, E3 +458007.505}
SPL {X  -165.650, Y  +553.092, Z    +0.000, E1   -30.157, E3 +458023.847}
SPL {X  -165.650, Y  +556.274, Z    +0.000, E1   -30.127, E3 +458035.102}
SPL {X  -165.650, Y  +560.243, Z    +0.000, E1   -30.214, E3 +458048.768}
SPL {X  -165.650, Y  +565.528, Z    +0.000, E1   -30.192, E3 +458067.460}
SPL {X  -165.650, Y  +570.048, Z    +0.000, E1   -30.238, E3 +458082.891}
SPL {X  -165.650, Y  +573.110, Z    +0.000, E1   -30.057, E3 +458094.876}
SPL {X  -165.650, Y  +576.497, Z    +0.000, E1   -30.234, E3 +458105.574}
SPL {X  -165.650, Y  +580.354, Z    +0.000, E1   -30.196, E3 +458119.589}
SPL {X  -165.650, Y  +585.053, Z    +0.000, E1   -30.090, E3 +458136.825}
ENDSPLINE

SPLINE
SPL {X  -165.650, Y  +484.445, Z    +0.000, E1   +32.277, E3 +458154.229}
SPL {X  -165.650, Y  +481.524, Z    +0.000, E1   +31.089, E3 +458171.680}
SPL {X  -165.650, Y  +478.014, Z    +0.000, E1   +30.826, E3 +458185.287}
SPL {X  -165.650, Y  +474.473, Z    +0.000, E1   +30.943, E3 +458196.612}
SPL {X  -165.650, Y  +470.376, Z    +0.000, E1   +30.888, E3 +458211.141}
SPL {X  -165.650, Y  +465.146, Z    +0.000, E1   +30.883, E3 +458229.071}
SPL {X  -165.650, Y  +461.106, Z    +0.000, E1   +30.916, E3 +458242.489}
SPL {X  -165.650, Y  +458.435, Z    +0.000, E1   +30.759, E3 +458252.697}
SPL {X  -165.650, Y  +454.220, Z    +0.000, E1   +30.954, E3 +458265.930}
SPL {X  -165.650, Y  +450.433, Z    +0.000, E1   +30.789, E3 +458279.895}
SPL {X  -165.650, Y  +447.097, Z    +0.000, E1   +30.843, E3 +458290.944}
SPL {X  -165.650, Y  +443.673, Z    +0.000, E1   +30.907, E3 +458302.251}
SPL {X  -165.650, Y  +440.976, Z    +0.000, E1   +30.719, E3 +458312.708}
SPL {X  -165.650, Y  +436.324, Z    +0.000, E1   +30.994, E3 +458326.994}
SPL {X  -165.650, Y  +432.765, Z    +0.000, E1   +30.831, E3 +458339.994}
SPL {X  -165.650, Y  +429.309, Z    +0.000, E1   +30.920, E3 +458351.335}
SPL {X  -165.650, Y  +424.918, Z    +0.000, E1   +30.862, E3 +458366.792}
SPL {X  -165.650, Y  +421.437, Z    +0.000, E1   +30.833, E3 +458378.761}
SPL {X  -165.650, Y  +418.489, Z    +0.000, E1   +30.835, E3 +458388.877}
SPL {X  -165.650, Y  +414.127, Z    +0.000, E1   +30.869, E3 +458403.786}
SPL {X  -165.650, Y  +408.547, Z    +0.000, E1   +30.964, E3 +458422.202}
SPL {X  -165.650, Y  +405.433, Z    +0.000, E1   +30.730, E3 +458434.179}
SPL {X  -165.650, Y  +402.516, Z    +0.000, E1   +30.874, E3 +458443.302}
SPL {X  -165.650, Y  +398.147, Z    +0.000, E1   +30.902, E3 +458458.180}
SPL {X  -165.650, Y  +394.694, Z    +0.000, E1   +30.805, E3 +458470.488}
SPL {X  -165.650, Y  +391.522, Z    +0.000, E1   +30.837, E3 +458481.169}
SPL {X  -165.650, Y  +387.533, Z    +0.000, E1   +30.858, E3 +458494.795}
SPL {X  -165.650, Y  +383.627, Z    +0.000, E1   +30.885, E3 +458507.856}
SPL {X  -165.650, Y  +379.886, Z    +0.000, E1   +30.887, E3 +458520.744}
SPL {X  -165.614, Y  +375.058, Z    +0.000, E1   +30.905, E3 +458537.197}
SPL {X  -165.492, Y  +371.263, Z    +0.000, E1   +30.913, E3 +458549.911}
SPL {X  -165.379, Y  +369.027, Z    +0.000, E1   +30.727, E3 +458558.849}
SPL {X  -165.167, Y  +365.866, Z    +0.000, E1   +30.741, E3 +458569.623}
SPL {X  -164.892, Y  +362.671, Z    +0.000, E1   +30.830, E3 +458579.948}
SPL {X  -164.570, Y  +359.612, Z    +0.000, E1   +30.773, E3 +458590.760}
SPL {X  -164.104, Y  +355.923, Z    +0.000, E1   +30.626, E3 +458604.477}
SPL {X  -163.573, Y  +352.353, Z    +0.000, E1   +30.451, E3 +458617.741}
SPL {X  -162.476, Y  +346.230, Z    +0.000, E1   +31.677, E3 +458630.322}
SPL {X  -152.976, Y  +314.952, Z    +0.000, E1   +38.607, E3 +458679.287}
SPL {X  -137.967, Y  +286.821, Z    +0.000, E1   +43.969, E3 +458722.509}
ENDSPLINE

SPLINE
SPL {X  -149.143, Y  +306.414, Z    +0.000, E1   +36.361, E3 +458773.641}
SPL {X  -164.268, Y  +357.145, Z    +0.000, E1   +15.880, E3 +458731.400}
SPL {X  -165.510, Y  +371.680, Z    +0.000, E1    +7.684, E3 +458734.402}
SPL {X  -165.628, Y  +375.818, Z    +0.000, E1    +5.016, E3 +458742.332}
SPL {X  -165.650, Y  +383.362, Z    +0.000, E1    +0.177, E3 +458723.366}
SPL {X  -165.650, Y  +383.923, Z    +0.000, E1    -0.215, E3 +458736.523}
SPL {X  -165.650, Y  +388.083, Z    +0.000, E1    -3.355, E3 +458735.386}
SPL {X  -165.650, Y  +393.983, Z    +0.000, E1    -8.501, E3 +458731.785}
SPL {X  -165.650, Y  +402.241, Z    +0.000, E1   -16.711, E3 +458726.296}
SPL {X  -165.650, Y  +416.345, Z    +0.000, E1   -29.511, E3 +458726.088}
SPL {X  -165.650, Y  +422.331, Z    +0.000, E1   -27.760, E3 +458751.587}
SPL {X  -165.650, Y  +441.276, Z    +0.000, E1   -37.343, E3 +458761.444}
SPL {X  -165.650, Y  +462.890, Z    +0.000, E1   -40.484, E3 +458795.527}
ENDSPLINE

SPLINE
SPL {X  -165.650, Y  +446.920, Z    +0.000, E1   -31.238, E3 +458807.853}
ENDSPLINE

SPLINE
SPL {X  -165.650, Y  +447.935, Z    +0.000, E1   -30.213, E3 +458818.141}
SPL {X  -165.650, Y  +451.020, Z    +0.000, E1   -30.224, E3 +458828.962}
SPL {X  -165.650, Y  +454.519, Z    +0.000, E1   -30.374, E3 +458840.144}
SPL {X  -165.650, Y  +456.542, Z    +0.000, E1   -29.986, E3 +458849.889}
SPL {X  -165.650, Y  +460.618, Z    +0.000, E1   -30.298, E3 +458862.209}
SPL {X  -165.650, Y  +463.853, Z    +0.000, E1   -30.103, E3 +458874.810}
SPL {X  -165.650, Y  +468.397, Z    +0.000, E1   -30.302, E3 +458889.614}
SPL {X  -165.650, Y  +472.566, Z    +0.000, E1   -30.124, E3 +458905.323}
SPL {X  -165.650, Y  +475.265, Z    +0.000, E1   -30.034, E3 +458915.361}
SPL {X  -165.650, Y  +477.862, Z    +0.000, E1   -30.319, E3 +458922.552}
SPL {X  -165.650, Y  +481.042, Z    +0.000, E1   -30.192, E3 +458934.812}
SPL {X  -165.650, Y  +485.236, Z    +0.000, E1   -30.294, E3 +458948.668}
SPL {X  -165.650, Y  +488.041, Z    +0.000, E1   -30.253, E3 +458958.789}
SPL {X  -165.650, Y  +491.281, Z    +0.000, E1   -30.148, E3 +458970.928}
SPL {X  -165.650, Y  +495.051, Z    +0.000, E1   -30.213, E3 +458983.736}
SPL {X  -165.650, Y  +499.546, Z    +0.000, E1   -30.283, E3 +458999.179}
SPL {X  -165.650, Y  +503.544, Z    +0.000, E1   -30.247, E3 +459013.247}
SPL {X  -165.650, Y  +506.344, Z    +0.000, E1   -30.129, E3 +459023.916}
SPL {X  -165.650, Y  +510.660, Z    +0.000, E1   -30.223, E3 +459038.619}
SPL {X  -165.650, Y  +514.670, Z    +0.000, E1   -30.278, E3 +459052.129}
SPL {X  -165.650, Y  +517.919, Z    +0.000, E1   -30.227, E3 +459063.989}
SPL {X  -165.650, Y  +521.521, Z    +0.000, E1   -30.210, E3 +459076.663}
SPL {X  -165.650, Y  +525.344, Z    +0.000, E1   -30.269, E3 +459089.770}
SPL {X  -165.650, Y  +528.152, Z    +0.000, E1   -29.991, E3 +459101.411}
SPL {X  -165.650, Y  +531.783, Z    +0.000, E1   -30.416, E3 +459111.303}
SPL {X  -165.650, Y  +534.115, Z    +0.000, E1   -30.089, E3 +459121.685}
SPL {X  -165.650, Y  +537.522, Z    +0.000, E1   -30.251, E3 +459132.600}
SPL {X  -165.650, Y  +540.621, Z    +0.000, E1   -30.014, E3 +459145.161}
SPL {X  -165.650, Y  +544.944, Z    +0.000, E1   -30.447, E3 +459157.360}
SPL {X  -165.650, Y  +547.199, Z    +0.000, E1   -30.132, E3 +459167.334}
SPL {X  -165.650, Y  +550.512, Z    +0.000, E1   -30.197, E3 +459178.660}
SPL {X  -165.650, Y  +553.852, Z    +0.000, E1   -30.156, E3 +459190.600}
SPL {X  -165.650, Y  +557.277, Z    +0.000, E1   -30.150, E3 +459202.775}
SPL {X  -165.650, Y  +561.168, Z    +0.000, E1   -30.194, E3 +459216.156}
SPL {X  -165.650, Y  +565.528, Z    +0.000, E1   -30.192, E3 +459231.639}
SPL {X  -165.650, Y  +570.048, Z    +0.000, E1   -30.238, E3 +459247.070}
SPL {X  -165.650, Y  +573.110, Z    +0.000, E1   -30.057, E3 +459259.055}
SPL {X  -165.650, Y  +577.587, Z    +0.000, E1   -30.270, E3 +459273.494}
SPL {X  -165.650, Y  +581.190, Z    +0.000, E1   -30.107, E3 +459287.133}
SPL {X  -165.650, Y  +585.053, Z    +0.000, E1   -30.090, E3 +459301.004}
ENDSPLINE

SPLINE
SPL {X  -165.650, Y  +484.445, Z    +0.000, E1   +32.277, E3 +459318.408}
SPL {X  -165.650, Y  +481.524, Z    +0.000, E1   +31.089, E3 +459335.859}
SPL {X  -165.650, Y  +478.014, Z    +0.000, E1   +30.826, E3 +459349.466}
SPL {X  -165.650, Y  +474.473, Z    +0.000, E1   +30.943, E3 +459360.791}
SPL {X  -165.650, Y  +470.376, Z    +0.000, E1   +30.888, E3 +459375.320}
SPL {X  -165.650, Y  +465.146, Z    +0.000, E1   +30.883, E3 +459393.250}
SPL {X  -165.650, Y  +461.106, Z    +0.000, E1   +30.916, E3 +459406.668}
SPL {X  -165.650, Y  +458.435, Z    +0.000, E1   +30.759, E3 +459416.876}
SPL {X  -165.650, Y  +454.220, Z    +0.000, E1   +30.954, E3 +459430.110}
SPL {X  -165.650, Y  +450.433, Z    +0.000, E1   +30.789, E3 +459444.074}
SPL {X  -165.650, Y  +447.097, Z    +0.000, E1   +30.843, E3 +459455.123}
SPL {X  -165.650, Y  +443.673, Z    +0.000, E1   +30.907, E3 +459466.430}
SPL {X  -165.650, Y  +440.976, Z    +0.000, E1   +30.719, E3 +459476.887}
SPL {X  -165.650, Y  +436.324, Z    +0.000, E1   +30.994, E3 +459491.174}
SPL {X  -165.650, Y  +432.765, Z    +0.000, E1   +30.831, E3 +459504.174}
SPL {X  -165.650, Y  +429.309, Z    +0.000, E1   +30.920, E3 +459515.514}
SPL {X  -165.650, Y  +424.918, Z    +0.000, E1   +30.862, E3 +459530.972}
SPL {X  -165.650, Y  +421.437, Z    +0.000, E1   +30.833, E3 +459542.940}
SPL {X  -165.650, Y  +417.366, Z    +0.000, E1   +30.879, E3 +459556.780}
SPL {X  -165.650, Y  +412.139, Z    +0.000, E1   +30.870, E3 +459574.730}
SPL {X  -165.650, Y  +406.834, Z    +0.000, E1   +30.919, E3 +459592.559}
SPL {X  -165.650, Y  +402.516, Z    +0.000, E1   +30.874, E3 +459607.481}
SPL {X  -165.650, Y  +398.147, Z    +0.000, E1   +30.902, E3 +459622.359}
SPL {X  -165.650, Y  +394.694, Z    +0.000, E1   +30.805, E3 +459634.667}
SPL {X  -165.650, Y  +391.522, Z    +0.000, E1   +30.837, E3 +459645.348}
SPL {X  -165.650, Y  +387.533, Z    +0.000, E1   +30.858, E3 +459658.975}
SPL {X  -165.650, Y  +383.627, Z    +0.000, E1   +30.885, E3 +459672.035}
SPL {X  -165.650, Y  +380.752, Z    +0.000, E1   +30.927, E3 +459681.549}
SPL {X  -165.648, Y  +377.739, Z    +0.000, E1   +30.835, E3 +459692.558}
SPL {X  -165.594, Y  +374.183, Z    +0.000, E1   +30.878, E3 +459704.395}
SPL {X  -165.492, Y  +371.263, Z    +0.000, E1   +30.913, E3 +459714.090}
SPL {X  -165.379, Y  +369.027, Z    +0.000, E1   +30.727, E3 +459723.029}
SPL {X  -165.167, Y  +365.866, Z    +0.000, E1   +30.741, E3 +459733.803}
SPL {X  -164.892, Y  +362.671, Z    +0.000, E1   +30.830, E3 +459744.127}
SPL {X  -164.570, Y  +359.612, Z    +0.000, E1   +30.773, E3 +459754.939}
SPL {X  -164.104, Y  +355.923, Z    +0.000, E1   +30.626, E3 +459768.656}
SPL {X  -163.573, Y  +352.353, Z    +0.000, E1   +30.451, E3 +459781.921}
SPL {X  -162.476, Y  +346.230, Z    +0.000, E1   +31.677, E3 +459794.501}
SPL {X  -152.976, Y  +314.952, Z    +0.000, E1   +38.607, E3 +459843.467}
SPL {X  -137.967, Y  +286.821, Z    +0.000, E1   +43.969, E3 +459886.688}
ENDSPLINE

SPLINE
SPL {X  -153.316, Y  +315.777, Z    +0.000, E1   +33.140, E3 +459929.315}
SPL {X  -164.446, Y  +358.564, Z    +0.000, E1   +15.149, E3 +459894.526}
SPL {X  -165.379, Y  +369.025, Z    +0.000, E1    +9.158, E3 +459900.251}
SPL {X  -165.612, Y  +374.969, Z    +0.000, E1    +5.630, E3 +459902.926}
SPL {X  -165.650, Y  +383.362, Z    +0.000, E1    +0.177, E3 +459887.545}
SPL {X  -165.650, Y  +383.923, Z    +0.000, E1    -0.215, E3 +459900.702}
SPL {X  -165.650, Y  +388.083, Z    +0.000, E1    -3.355, E3 +459899.566}
SPL {X  -165.650, Y  +393.983, Z    +0.000, E1    -8.501, E3 +459895.964}
SPL {X  -165.650, Y  +402.241, Z    +0.000, E1   -16.711, E3 +459890.476}
SPL {X  -165.650, Y  +416.345, Z    +0.000, E1   -29.511, E3 +459890.267}
SPL {X  -165.650, Y  +422.331, Z    +0.000, E1   -27.760, E3 +459915.767}
SPL {X  -165.650, Y  +441.276, Z    +0.000, E1   -37.343, E3 +459925.624}
SPL {X  -165.650, Y  +462.890, Z    +0.000, E1   -40.484, E3 +459959.706}
ENDSPLINE

SPLINE
SPL {X  -165.650, Y  +446.920, Z    +0.000, E1   -31.238, E3 +459972.032}
ENDSPLINE

SPLINE
SPL {X  -165.650, Y  +447.935, Z    +0.000, E1   -30.213, E3 +459982.320}
SPL {X  -165.650, Y  +451.020, Z    +0.000, E1   -30.224, E3 +459993.141}
SPL {X  -165.650, Y  +454.519, Z    +0.000, E1   -30.374, E3 +460004.323}
SPL {X  -165.650, Y  +456.542, Z    +0.000, E1   -29.986, E3 +460014.068}
SPL {X  -165.650, Y  +460.618, Z    +0.000, E1   -30.298, E3 +460026.388}
SPL {X  -165.650, Y  +463.853, Z    +0.000, E1   -30.103, E3 +460038.989}
SPL {X  -165.650, Y  +467.246, Z    +0.000, E1   -30.279, E3 +460049.719}
SPL {X  -165.650, Y  +469.780, Z    +0.000, E1   -30.237, E3 +460058.844}
SPL {X  -165.650, Y  +472.566, Z    +0.000, E1   -30.124, E3 +460069.502}
SPL {X  -165.650, Y  +476.540, Z    +0.000, E1   -30.193, E3 +460083.046}
SPL {X  -165.650, Y  +480.320, Z    +0.000, E1   -30.163, E3 +460096.524}
SPL {X  -165.650, Y  +484.477, Z    +0.000, E1   -30.274, E3 +460110.413}
SPL {X  -165.650, Y  +488.041, Z    +0.000, E1   -30.253, E3 +460122.968}
SPL {X  -165.650, Y  +491.281, Z    +0.000, E1   -30.148, E3 +460135.107}
SPL {X  -165.650, Y  +495.051, Z    +0.000, E1   -30.213, E3 +460147.915}
SPL {X  -165.650, Y  +498.418, Z    +0.000, E1   -30.282, E3 +460159.208}
SPL {X  -165.650, Y  +500.833, Z    +0.000, E1   -30.191, E3 +460168.257}
SPL {X  -165.650, Y  +504.246, Z    +0.000, E1   -30.231, E3 +460180.123}
SPL {X  -165.650, Y  +507.017, Z    +0.000, E1   -30.108, E3 +460190.532}
SPL {X  -165.650, Y  +510.660, Z    +0.000, E1   -30.223, E3 +460202.799}
SPL {X  -165.650, Y  +515.918, Z    +0.000, E1   -30.316, E3 +460220.607}
SPL {X  -165.650, Y  +520.621, Z    +0.000, E1   -30.198, E3 +460237.892}
SPL {X  -165.650, Y  +525.344, Z    +0.000, E1   -30.269, E3 +460253.949}
SPL {X  -165.650, Y  +528.152, Z    +0.000, E1   -29.991, E3 +460265.590}
SPL {X  -165.650, Y  +531.783, Z    +0.000, E1   -30.416, E3 +460275.482}
SPL {X  -165.650, Y  +534.115, Z    +0.000, E1   -30.089, E3 +460285.864}
SPL {X  -165.650, Y  +538.363, Z    +0.000, E1   -30.232, E3 +460300.034}
SPL {X  -165.650, Y  +543.650, Z    +0.000, E1   -30.281, E3 +460318.254}
SPL {X  -165.650, Y  +547.199, Z    +0.000, E1   -30.132, E3 +460331.513}
SPL {X  -165.650, Y  +550.512, Z    +0.000, E1   -30.197, E3 +460342.839}
SPL {X  -165.650, Y  +554.908, Z    +0.000, E1   -30.180, E3 +460358.500}
SPL {X  -165.650, Y  +560.243, Z    +0.000, E1   -30.214, E3 +460377.126}
SPL {X  -165.650, Y  +565.528, Z    +0.000, E1   -30.192, E3 +460395.818}
SPL {X  -165.650, Y  +570.048, Z    +0.000, E1   -30.238, E3 +460411.249}
SPL {X  -165.650, Y  +573.110, Z    +0.000, E1   -30.057, E3 +460423.234}
SPL {X  -165.650, Y  +577.587, Z    +0.000, E1   -30.270, E3 +460437.673}
SPL {X  -165.650, Y  +581.190, Z    +0.000, E1   -30.107, E3 +460451.313}
SPL {X  -165.650, Y  +585.096, Z    +0.000, E1   -30.203, E3 +460464.499}
ENDSPLINE

SPLINE
SPL {X  -165.650, Y  +584.346, Z    +0.000, E1   -28.397, E3 +460473.846}
SPL {X  -165.650, Y  +484.445, Z    +0.000, E1   +32.277, E3 +460482.587}
SPL {X  -165.650, Y  +481.524, Z    +0.000, E1   +31.089, E3 +460500.038}
SPL {X  -165.650, Y  +478.014, Z    +0.000, E1   +30.826, E3 +460513.645}
SPL {X  -165.650, Y  +474.473, Z    +0.000, E1   +30.943, E3 +460524.970}
SPL {X  -165.650, Y  +471.826, Z    +0.000, E1   +30.770, E3 +460535.153}
SPL {X  -165.650, Y  +467.753, Z    +0.000, E1   +30.878, E3 +460548.527}
SPL {X  -165.650, Y  +463.837, Z    +0.000, E1   +30.924, E3 +460561.461}
SPL {X  -165.650, Y  +461.106, Z    +0.000, E1   +30.916, E3 +460570.848}
SPL {X  -165.650, Y  +457.156, Z    +0.000, E1   +30.860, E3 +460584.924}
SPL {X  -165.650, Y  +453.156, Z    +0.000, E1   +30.934, E3 +460597.898}
SPL {X  -165.650, Y  +450.433, Z    +0.000, E1   +30.789, E3 +460608.253}
SPL {X  -165.650, Y  +447.097, Z    +0.000, E1   +30.843, E3 +460619.302}
SPL {X  -165.650, Y  +443.673, Z    +0.000, E1   +30.907, E3 +460630.610}
SPL {X  -165.650, Y  +439.486, Z    +0.000, E1   +30.857, E3 +460645.419}
SPL {X  -165.650, Y  +434.043, Z    +0.000, E1   +30.950, E3 +460663.435}
SPL {X  -165.650, Y  +430.419, Z    +0.000, E1   +30.895, E3 +460675.938}
SPL {X  -165.650, Y  +427.340, Z    +0.000, E1   +30.870, E3 +460686.765}
SPL {X  -165.650, Y  +422.641, Z    +0.000, E1   +30.884, E3 +460702.854}
SPL {X  -165.650, Y  +417.366, Z    +0.000, E1   +30.879, E3 +460720.959}
SPL {X  -165.650, Y  +412.139, Z    +0.000, E1   +30.870, E3 +460738.909}
SPL {X  -165.650, Y  +406.834, Z    +0.000, E1   +30.919, E3 +460756.738}
SPL {X  -165.650, Y  +402.516, Z    +0.000, E1   +30.874, E3 +460771.660}
SPL {X  -165.650, Y  +398.147, Z    +0.000, E1   +30.902, E3 +460786.538}
SPL {X  -165.650, Y  +394.694, Z    +0.000, E1   +30.805, E3 +460798.847}
SPL {X  -165.650, Y  +391.522, Z    +0.000, E1   +30.837, E3 +460809.527}
SPL {X  -165.650, Y  +387.533, Z    +0.000, E1   +30.858, E3 +460823.154}
SPL {X  -165.650, Y  +383.627, Z    +0.000, E1   +30.885, E3 +460836.214}
SPL {X  -165.650, Y  +380.752, Z    +0.000, E1   +30.927, E3 +460845.728}
SPL {X  -165.648, Y  +377.739, Z    +0.000, E1   +30.835, E3 +460856.737}
SPL {X  -165.594, Y  +374.183, Z    +0.000, E1   +30.878, E3 +460868.574}
SPL {X  -165.492, Y  +371.263, Z    +0.000, E1   +30.913, E3 +460878.269}
SPL {X  -165.379, Y  +369.027, Z    +0.000, E1   +30.727, E3 +460887.208}
SPL {X  -165.167, Y  +365.866, Z    +0.000, E1   +30.741, E3 +460897.982}
SPL {X  -164.892, Y  +362.671, Z    +0.000, E1   +30.830, E3 +460908.306}
SPL {X  -164.570, Y  +359.612, Z    +0.000, E1   +30.773, E3 +460919.118}
SPL {X  -164.104, Y  +355.923, Z    +0.000, E1   +30.626, E3 +460932.835}
SPL {X  -163.573, Y  +352.353, Z    +0.000, E1   +30.451, E3 +460946.100}
SPL {X  -162.476, Y  +346.230, Z    +0.000, E1   +31.677, E3 +460958.680}
SPL {X  -152.976, Y  +314.952, Z    +0.000, E1   +38.607, E3 +461007.646}
SPL {X  -137.967, Y  +286.821, Z    +0.000, E1   +43.969, E3 +461050.867}
ENDSPLINE

SPLINE
SPL {X  -153.316, Y  +315.777, Z    +0.000, E1   +33.140, E3 +461093.494}
SPL {X  -164.446, Y  +358.564, Z    +0.000, E1   +15.149, E3 +461058.705}
SPL {X  -165.379, Y  +369.025, Z    +0.000, E1    +9.158, E3 +461064.430}
SPL {X  -165.612, Y  +374.969, Z    +0.000, E1    +5.630, E3 +461067.105}
SPL {X  -165.650, Y  +383.362, Z    +0.000, E1    +0.177, E3 +461051.724}
SPL {X  -165.650, Y  +383.923, Z    +0.000, E1    -0.215, E3 +461064.881}
SPL {X  -165.650, Y  +388.083, Z    +0.000, E1    -3.355, E3 +461063.745}
SPL {X  -165.650, Y  +393.983, Z    +0.000, E1    -8.501, E3 +461060.143}
SPL {X  -165.650, Y  +402.241, Z    +0.000, E1   -16.711, E3 +461054.655}
SPL {X  -165.650, Y  +416.345, Z    +0.000, E1   -29.511, E3 +461054.447}
SPL {X  -165.650, Y  +422.331, Z    +0.000, E1   -27.760, E3 +461079.946}
SPL {X  -165.650, Y  +441.276, Z    +0.000, E1   -37.343, E3 +461089.803}
SPL {X  -165.650, Y  +462.890, Z    +0.000, E1   -40.484, E3 +461123.886}
ENDSPLINE

SPLINE
SPL {X  -165.650, Y  +446.920, Z    +0.000, E1   -31.238, E3 +461136.211}
ENDSPLINE

SPLINE
SPL {X  -165.650, Y  +447.935, Z    +0.000, E1   -30.213, E3 +461146.499}
SPL {X  -165.650, Y  +451.020, Z    +0.000, E1   -30.224, E3 +461157.320}
SPL {X  -165.650, Y  +454.519, Z    +0.000, E1   -30.374, E3 +461168.502}
SPL {X  -165.650, Y  +457.429, Z    +0.000, E1   -30.029, E3 +461181.204}
SPL {X  -165.650, Y  +461.678, Z    +0.000, E1   -30.426, E3 +461193.328}
SPL {X  -165.650, Y  +463.853, Z    +0.000, E1   -30.103, E3 +461203.168}
SPL {X  -165.650, Y  +468.397, Z    +0.000, E1   -30.302, E3 +461217.972}
SPL {X  -165.650, Y  +472.566, Z    +0.000, E1   -30.124, E3 +461233.681}
SPL {X  -165.650, Y  +476.540, Z    +0.000, E1   -30.193, E3 +461247.225}
SPL {X  -165.650, Y  +481.042, Z    +0.000, E1   -30.192, E3 +461263.171}
SPL {X  -165.650, Y  +485.236, Z    +0.000, E1   -30.294, E3 +461277.026}
SPL {X  -165.650, Y  +489.057, Z    +0.000, E1   -30.341, E3 +461290.232}
SPL {X  -165.650, Y  +491.647, Z    +0.000, E1   -29.894, E3 +461302.165}
SPL {X  -165.650, Y  +495.051, Z    +0.000, E1   -30.213, E3 +461312.094}
SPL {X  -165.650, Y  +498.418, Z    +0.000, E1   -30.282, E3 +461323.387}
SPL {X  -165.650, Y  +502.421, Z    +0.000, E1   -30.263, E3 +461337.745}
SPL {X  -165.650, Y  +506.344, Z    +0.000, E1   -30.129, E3 +461352.274}
SPL {X  -165.650, Y  +509.866, Z    +0.000, E1   -30.236, E3 +461363.943}
SPL {X  -165.650, Y  +513.685, Z    +0.000, E1   -30.234, E3 +461377.440}
SPL {X  -165.650, Y  +517.919, Z    +0.000, E1   -30.227, E3 +461392.347}
SPL {X  -165.650, Y  +521.521, Z    +0.000, E1   -30.210, E3 +461405.022}
SPL {X  -165.650, Y  +525.344, Z    +0.000, E1   -30.269, E3 +461418.128}
SPL {X  -165.650, Y  +528.152, Z    +0.000, E1   -29.991, E3 +461429.769}
SPL {X  -165.650, Y  +531.783, Z    +0.000, E1   -30.416, E3 +461439.662}
SPL {X  -165.650, Y  +534.115, Z    +0.000, E1   -30.089, E3 +461450.044}
SPL {X  -165.650, Y  +537.522, Z    +0.000, E1   -30.251, E3 +461460.958}
SPL {X  -165.650, Y  +540.621, Z    +0.000, E1   -30.014, E3 +461473.519}
SPL {X  -165.650, Y  +544.944, Z    +0.000, E1   -30.447, E3 +461485.718}
SPL {X  -165.650, Y  +548.549, Z    +0.000, E1   -30.216, E3 +461500.042}
SPL {X  -165.650, Y  +553.092, Z    +0.000, E1   -30.157, E3 +461516.384}
SPL {X  -165.650, Y  +556.274, Z    +0.000, E1   -30.127, E3 +461527.639}
SPL {X  -165.650, Y  +560.243, Z    +0.000, E1   -30.214, E3 +461541.305}
SPL {X  -165.650, Y  +565.528, Z    +0.000, E1   -30.192, E3 +461559.997}
SPL {X  -165.650, Y  +570.048, Z    +0.000, E1   -30.238, E3 +461575.428}
SPL {X  -165.650, Y  +573.110, Z    +0.000, E1   -30.057, E3 +461587.413}
SPL {X  -165.650, Y  +577.587, Z    +0.000, E1   -30.270, E3 +461601.852}
SPL {X  -165.650, Y  +581.190, Z    +0.000, E1   -30.107, E3 +461615.492}
SPL {X  -165.650, Y  +585.053, Z    +0.000, E1   -30.090, E3 +461629.362}
ENDSPLINE

SPLINE
SPL {X  -165.650, Y  +484.445, Z    +0.000, E1   +32.277, E3 +461646.766}
SPL {X  -165.650, Y  +481.524, Z    +0.000, E1   +31.089, E3 +461664.217}
SPL {X  -165.650, Y  +478.014, Z    +0.000, E1   +30.826, E3 +461677.824}
SPL {X  -165.650, Y  +474.473, Z    +0.000, E1   +30.943, E3 +461689.149}
SPL {X  -165.650, Y  +471.826, Z    +0.000, E1   +30.770, E3 +461699.332}
SPL {X  -165.650, Y  +467.753, Z    +0.000, E1   +30.878, E3 +461712.706}
SPL {X  -165.650, Y  +463.837, Z    +0.000, E1   +30.924, E3 +461725.640}
SPL {X  -165.650, Y  +461.106, Z    +0.000, E1   +30.916, E3 +461735.027}
SPL {X  -165.650, Y  +458.435, Z    +0.000, E1   +30.759, E3 +461745.235}
SPL {X  -165.650, Y  +454.220, Z    +0.000, E1   +30.954, E3 +461758.468}
SPL {X  -165.650, Y  +450.433, Z    +0.000, E1   +30.789, E3 +461772.432}
SPL {X  -165.650, Y  +447.097, Z    +0.000, E1   +30.843, E3 +461783.481}
SPL {X  -165.650, Y  +443.673, Z    +0.000, E1   +30.907, E3 +461794.789}
SPL {X  -165.650, Y  +440.976, Z    +0.000, E1   +30.719, E3 +461805.245}
SPL {X  -165.650, Y  +436.324, Z    +0.000, E1   +30.994, E3 +461819.532}
SPL {X  -165.650, Y  +432.765, Z    +0.000, E1   +30.831, E3 +461832.532}
SPL {X  -165.650, Y  +429.309, Z    +0.000, E1   +30.920, E3 +461843.873}
SPL {X  -165.650, Y  +424.918, Z    +0.000, E1   +30.862, E3 +461859.330}
SPL {X  -165.650, Y  +421.437, Z    +0.000, E1   +30.833, E3 +461871.298}
SPL {X  -165.650, Y  +417.366, Z    +0.000, E1   +30.879, E3 +461885.139}
SPL {X  -165.650, Y  +413.181, Z    +0.000, E1   +30.815, E3 +461899.736}
SPL {X  -165.650, Y  +408.547, Z    +0.000, E1   +30.964, E3 +461914.739}
SPL {X  -165.650, Y  +403.421, Z    +0.000, E1   +30.863, E3 +461932.957}
SPL {X  -165.650, Y  +398.147, Z    +0.000, E1   +30.902, E3 +461950.717}
SPL {X  -165.650, Y  +394.694, Z    +0.000, E1   +30.805, E3 +461963.026}
SPL {X  -165.650, Y  +391.522, Z    +0.000, E1   +30.837, E3 +461973.707}
SPL {X  -165.650, Y  +387.533, Z    +0.000, E1   +30.858, E3 +461987.333}
SPL {X  -165.650, Y  +383.627, Z    +0.000, E1   +30.885, E3 +462000.393}
SPL {X  -165.650, Y  +379.886, Z    +0.000, E1   +30.887, E3 +462013.281}
SPL {X  -165.614, Y  +375.058, Z    +0.000, E1   +30.905, E3 +462029.734}
SPL {X  -165.492, Y  +371.263, Z    +0.000, E1   +30.913, E3 +462042.448}
SPL {X  -165.379, Y  +369.027, Z    +0.000, E1   +30.727, E3 +462051.387}
SPL {X  -165.167, Y  +365.866, Z    +0.000, E1   +30.741, E3 +462062.161}
SPL {X  -164.892, Y  +362.671, Z    +0.000, E1   +30.830, E3 +462072.485}
SPL {X  -164.570, Y  +359.612, Z    +0.000, E1   +30.773, E3 +462083.297}
SPL {X  -164.104, Y  +355.923, Z    +0.000, E1   +30.626, E3 +462097.014}
SPL {X  -163.573, Y  +352.353, Z    +0.000, E1   +30.451, E3 +462110.279}
SPL {X  -162.476, Y  +346.230, Z    +0.000, E1   +31.677, E3 +462122.860}
SPL {X  -152.976, Y  +314.952, Z    +0.000, E1   +38.607, E3 +462171.825}
SPL {X  -137.967, Y  +286.821, Z    +0.000, E1   +43.969, E3 +462215.046}
ENDSPLINE

SPLINE
SPL {X  -153.316, Y  +315.777, Z    +0.000, E1   +33.140, E3 +462257.673}
SPL {X  -164.446, Y  +358.564, Z    +0.000, E1   +15.149, E3 +462222.884}
SPL {X  -165.510, Y  +371.680, Z    +0.000, E1    +7.684, E3 +462226.940}
SPL {X  -165.628, Y  +375.818, Z    +0.000, E1    +5.016, E3 +462234.869}
SPL {X  -165.650, Y  +383.362, Z    +0.000, E1    +0.177, E3 +462215.903}
SPL {X  -165.650, Y  +383.923, Z    +0.000, E1    -0.215, E3 +462229.060}
SPL {X  -165.650, Y  +388.083, Z    +0.000, E1    -3.355, E3 +462227.924}
SPL {X  -165.650, Y  +393.983, Z    +0.000, E1    -8.501, E3 +462224.322}
SPL {X  -165.650, Y  +402.241, Z    +0.000, E1   -16.711, E3 +462218.834}
SPL {X  -165.650, Y  +414.811, Z    +0.000, E1   -28.314, E3 +462218.364}
SPL {X  -165.650, Y  +423.479, Z    +0.000, E1   -29.012, E3 +462242.293}
SPL {X  -165.650, Y  +441.276, Z    +0.000, E1   -37.343, E3 +462253.982}
SPL {X  -165.650, Y  +462.890, Z    +0.000, E1   -40.484, E3 +462288.065}
ENDSPLINE

SPLINE
SPL {X  -165.650, Y  +446.920, Z    +0.000, E1   -31.238, E3 +462300.391}
ENDSPLINE

SPLINE
SPL {X  -165.650, Y  +447.935, Z    +0.000, E1   -30.213, E3 +462310.678}
SPL {X  -165.650, Y  +451.020, Z    +0.000, E1   -30.224, E3 +462321.499}
SPL {X  -165.650, Y  +454.519, Z    +0.000, E1   -30.374, E3 +462332.681}
SPL {X  -165.650, Y  +456.542, Z    +0.000, E1   -29.986, E3 +462342.426}
SPL {X  -165.650, Y  +460.618, Z    +0.000, E1   -30.298, E3 +462354.746}
SPL {X  -165.650, Y  +463.853, Z    +0.000, E1   -30.103, E3 +462367.347}
SPL {X  -165.650, Y  +468.397, Z    +0.000, E1   -30.302, E3 +462382.151}
SPL {X  -165.650, Y  +472.566, Z    +0.000, E1   -30.124, E3 +462397.860}
SPL {X  -165.650, Y  +475.265, Z    +0.000, E1   -30.034, E3 +462407.898}
SPL {X  -165.650, Y  +477.862, Z    +0.000, E1   -30.319, E3 +462415.089}
SPL {X  -165.650, Y  +481.042, Z    +0.000, E1   -30.192, E3 +462427.350}
SPL {X  -165.650, Y  +485.236, Z    +0.000, E1   -30.294, E3 +462441.205}
SPL {X  -165.650, Y  +488.041, Z    +0.000, E1   -30.253, E3 +462451.327}
SPL {X  -165.650, Y  +491.281, Z    +0.000, E1   -30.148, E3 +462463.465}
SPL {X  -165.650, Y  +495.051, Z    +0.000, E1   -30.213, E3 +462476.273}
SPL {X  -165.650, Y  +499.546, Z    +0.000, E1   -30.283, E3 +462491.716}
SPL {X  -165.650, Y  +503.544, Z    +0.000, E1   -30.247, E3 +462505.785}
SPL {X  -165.650, Y  +506.344, Z    +0.000, E1   -30.129, E3 +462516.453}
SPL {X  -165.650, Y  +510.660, Z    +0.000, E1   -30.223, E3 +462531.157}
SPL {X  -165.650, Y  +514.670, Z    +0.000, E1   -30.278, E3 +462544.666}
SPL {X  -165.650, Y  +517.919, Z    +0.000, E1   -30.227, E3 +462556.526}
SPL {X  -165.650, Y  +521.521, Z    +0.000, E1   -30.210, E3 +462569.201}
SPL {X  -165.650, Y  +525.344, Z    +0.000, E1   -30.269, E3 +462582.307}
SPL {X  -165.650, Y  +528.152, Z    +0.000, E1   -29.991, E3 +462593.948}
SPL {X  -165.650, Y  +531.783, Z    +0.000, E1   -30.416, E3 +462603.841}
SPL {X  -165.650, Y  +534.115, Z    +0.000, E1   -30.089, E3 +462614.223}
SPL {X  -165.650, Y  +537.522, Z    +0.000, E1   -30.251, E3 +462625.137}
SPL {X  -165.650, Y  +540.621, Z    +0.000, E1   -30.014, E3 +462637.698}
SPL {X  -165.650, Y  +544.944, Z    +0.000, E1   -30.447, E3 +462649.898}
SPL {X  -165.650, Y  +547.199, Z    +0.000, E1   -30.132, E3 +462659.871}
SPL {X  -165.650, Y  +550.512, Z    +0.000, E1   -30.197, E3 +462671.197}
SPL {X  -165.650, Y  +553.852, Z    +0.000, E1   -30.156, E3 +462683.138}
SPL {X  -165.650, Y  +557.277, Z    +0.000, E1   -30.150, E3 +462695.312}
SPL {X  -165.650, Y  +561.168, Z    +0.000, E1   -30.194, E3 +462708.694}
SPL {X  -165.650, Y  +564.449, Z    +0.000, E1   -30.167, E3 +462720.377}
SPL {X  -165.650, Y  +566.935, Z    +0.000, E1   -30.135, E3 +462729.282}
SPL {X  -165.650, Y  +570.048, Z    +0.000, E1   -30.238, E3 +462739.607}
SPL {X  -165.650, Y  +573.110, Z    +0.000, E1   -30.057, E3 +462751.592}
SPL {X  -165.650, Y  +577.587, Z    +0.000, E1   -30.270, E3 +462766.031}
SPL {X  -165.650, Y  +581.190, Z    +0.000, E1   -30.107, E3 +462779.671}
SPL {X  -165.650, Y  +585.053, Z    +0.000, E1   -30.090, E3 +462793.541}
ENDSPLINE

SPLINE
SPL {X  -165.650, Y  +484.445, Z    +0.000, E1   +32.277, E3 +462810.945}
SPL {X  -165.650, Y  +481.524, Z    +0.000, E1   +31.089, E3 +462828.396}
SPL {X  -165.650, Y  +478.014, Z    +0.000, E1   +30.826, E3 +462842.004}
SPL {X  -165.650, Y  +474.473, Z    +0.000, E1   +30.943, E3 +462853.328}
SPL {X  -165.650, Y  +471.826, Z    +0.000, E1   +30.770, E3 +462863.511}
SPL {X  -165.650, Y  +467.753, Z    +0.000, E1   +30.878, E3 +462876.885}
SPL {X  -165.650, Y  +463.837, Z    +0.000, E1   +30.924, E3 +462889.819}
SPL {X  -165.650, Y  +461.106, Z    +0.000, E1   +30.916, E3 +462899.206}
SPL {X  -165.650, Y  +458.435, Z    +0.000, E1   +30.759, E3 +462909.414}
SPL {X  -165.650, Y  +454.220, Z    +0.000, E1   +30.954, E3 +462922.647}
SPL {X  -165.650, Y  +450.433, Z    +0.000, E1   +30.789, E3 +462936.612}
SPL {X  -165.650, Y  +447.097, Z    +0.000, E1   +30.843, E3 +462947.660}
SPL {X  -165.650, Y  +443.673, Z    +0.000, E1   +30.907, E3 +462958.968}
SPL {X  -165.650, Y  +440.976, Z    +0.000, E1   +30.719, E3 +462969.424}
SPL {X  -165.650, Y  +437.973, Z    +0.000, E1   +30.928, E3 +462978.297}
SPL {X  -165.650, Y  +434.043, Z    +0.000, E1   +30.950, E3 +462991.793}
SPL {X  -165.650, Y  +430.419, Z    +0.000, E1   +30.895, E3 +463004.296}
SPL {X  -165.650, Y  +427.340, Z    +0.000, E1   +30.870, E3 +463015.123}
SPL {X  -165.650, Y  +422.641, Z    +0.000, E1   +30.884, E3 +463031.212}
SPL {X  -165.650, Y  +418.489, Z    +0.000, E1   +30.835, E3 +463045.594}
SPL {X  -165.650, Y  +414.127, Z    +0.000, E1   +30.869, E3 +463060.503}
SPL {X  -165.650, Y  +408.547, Z    +0.000, E1   +30.964, E3 +463078.918}
SPL {X  -165.650, Y  +405.433, Z    +0.000, E1   +30.730, E3 +463090.895}
SPL {X  -165.650, Y  +402.516, Z    +0.000, E1   +30.874, E3 +463100.018}
SPL {X  -165.650, Y  +398.147, Z    +0.000, E1   +30.902, E3 +463114.896}
SPL {X  -165.650, Y  +394.694, Z    +0.000, E1   +30.805, E3 +463127.205}
SPL {X  -165.650, Y  +391.522, Z    +0.000, E1   +30.837, E3 +463137.886}
SPL {X  -165.650, Y  +387.533, Z    +0.000, E1   +30.858, E3 +463151.512}
SPL {X  -165.650, Y  +383.627, Z    +0.000, E1   +30.885, E3 +463164.572}
SPL {X  -165.650, Y  +379.886, Z    +0.000, E1   +30.887, E3 +463177.460}
SPL {X  -165.614, Y  +375.058, Z    +0.000, E1   +30.905, E3 +463193.913}
SPL {X  -165.492, Y  +371.263, Z    +0.000, E1   +30.913, E3 +463206.627}
SPL {X  -165.379, Y  +369.027, Z    +0.000, E1   +30.727, E3 +463215.566}
SPL {X  -165.167, Y  +365.866, Z    +0.000, E1   +30.741, E3 +463226.340}
SPL {X  -164.892, Y  +362.671, Z    +0.000, E1   +30.830, E3 +463236.664}
SPL {X  -164.570, Y  +359.612, Z    +0.000, E1   +30.773, E3 +463247.477}
SPL {X  -164.104, Y  +355.923, Z    +0.000, E1   +30.626, E3 +463261.193}
SPL {X  -163.573, Y  +352.353, Z    +0.000, E1   +30.451, E3 +463274.458}
SPL {X  -162.976, Y  +348.856, Z    +0.000, E1   +30.757, E3 +463284.382}
SPL {X  -161.497, Y  +341.640, Z    +0.000, E1   +33.276, E3 +463291.659}
SPL {X  -152.976, Y  +314.952, Z    +0.000, E1   +38.607, E3 +463336.004}
SPL {X  -137.967, Y  +286.821, Z    +0.000, E1   +43.969, E3 +463379.225}
ENDSPLINE

SPLINE
SPL {X  -149.143, Y  +306.414, Z    +0.000, E1   +36.361, E3 +463430.357}
SPL {X  -164.268, Y  +357.145, Z    +0.000, E1   +15.880, E3 +463388.117}
SPL {X  -165.379, Y  +369.025, Z    +0.000, E1    +9.158, E3 +463392.788}
SPL {X  -165.612, Y  +374.969, Z    +0.000, E1    +5.630, E3 +463395.464}
SPL {X  -165.650, Y  +383.362, Z    +0.000, E1    +0.177, E3 +463380.082}
SPL {X  -165.650, Y  +383.923, Z    +0.000, E1    -0.215, E3 +463393.239}
SPL {X  -165.650, Y  +388.083, Z    +0.000, E1    -3.355, E3 +463392.103}
SPL {X  -165.650, Y  +393.983, Z    +0.000, E1    -8.501, E3 +463388.501}
SPL {X  -165.650, Y  +402.241, Z    +0.000, E1   -16.711, E3 +463383.013}
SPL {X  -165.650, Y  +416.345, Z    +0.000, E1   -29.511, E3 +463382.805}
SPL {X  -165.650, Y  +422.331, Z    +0.000, E1   -27.760, E3 +463408.304}
SPL {X  -165.650, Y  +441.276, Z    +0.000, E1   -37.343, E3 +463418.161}
SPL {X  -165.650, Y  +462.890, Z    +0.000, E1   -40.484, E3 +463452.244}
ENDSPLINE

SPLINE
SPL {X  -165.650, Y  +446.920, Z    +0.000, E1   -31.238, E3 +463464.570}
ENDSPLINE

SPLINE
SPL {X  -165.650, Y  +447.935, Z    +0.000, E1   -30.213, E3 +463474.858}
SPL {X  -165.650, Y  +451.020, Z    +0.000, E1   -30.224, E3 +463485.678}
SPL {X  -165.650, Y  +454.519, Z    +0.000, E1   -30.374, E3 +463496.860}
SPL {X  -165.650, Y  +456.542, Z    +0.000, E1   -29.986, E3 +463506.605}
SPL {X  -165.650, Y  +460.618, Z    +0.000, E1   -30.298, E3 +463518.926}
SPL {X  -165.650, Y  +463.853, Z    +0.000, E1   -30.103, E3 +463531.526}
SPL {X  -165.650, Y  +468.397, Z    +0.000, E1   -30.302, E3 +463546.330}
SPL {X  -165.650, Y  +472.566, Z    +0.000, E1   -30.124, E3 +463562.039}
SPL {X  -165.650, Y  +476.540, Z    +0.000, E1   -30.193, E3 +463575.584}
SPL {X  -165.650, Y  +480.320, Z    +0.000, E1   -30.163, E3 +463589.061}
SPL {X  -165.650, Y  +484.477, Z    +0.000, E1   -30.274, E3 +463602.951}
SPL {X  -165.650, Y  +488.041, Z    +0.000, E1   -30.253, E3 +463615.506}
SPL {X  -165.650, Y  +491.281, Z    +0.000, E1   -30.148, E3 +463627.644}
SPL {X  -165.650, Y  +495.051, Z    +0.000, E1   -30.213, E3 +463640.452}
SPL {X  -165.650, Y  +499.546, Z    +0.000, E1   -30.283, E3 +463655.895}
SPL {X  -165.650, Y  +503.544, Z    +0.000, E1   -30.247, E3 +463669.964}
SPL {X  -165.650, Y  +506.344, Z    +0.000, E1   -30.129, E3 +463680.632}
SPL {X  -165.650, Y  +509.866, Z    +0.000, E1   -30.236, E3 +463692.302}
SPL {X  -165.650, Y  +513.685, Z    +0.000, E1   -30.234, E3 +463705.798}
SPL {X  -165.650, Y  +517.919, Z    +0.000, E1   -30.227, E3 +463720.705}
SPL {X  -165.650, Y  +521.521, Z    +0.000, E1   -30.210, E3 +463733.380}
SPL {X  -165.650, Y  +525.344, Z    +0.000, E1   -30.269, E3 +463746.486}
SPL {X  -165.650, Y  +528.152, Z    +0.000, E1   -29.991, E3 +463758.127}
SPL {X  -165.650, Y  +531.783, Z    +0.000, E1   -30.416, E3 +463768.020}
SPL {X  -165.650, Y  +534.115, Z    +0.000, E1   -30.089, E3 +463778.402}
SPL {X  -165.650, Y  +537.522, Z    +0.000, E1   -30.251, E3 +463789.316}
SPL {X  -165.650, Y  +540.621, Z    +0.000, E1   -30.014, E3 +463801.877}
SPL {X  -165.650, Y  +544.944, Z    +0.000, E1   -30.447, E3 +463814.077}
SPL {X  -165.650, Y  +547.199, Z    +0.000, E1   -30.132, E3 +463824.050}
SPL {X  -165.650, Y  +550.512, Z    +0.000, E1   -30.197, E3 +463835.376}
SPL {X  -165.650, Y  +553.852, Z    +0.000, E1   -30.156, E3 +463847.317}
SPL {X  -165.650, Y  +557.277, Z    +0.000, E1   -30.150, E3 +463859.491}
SPL {X  -165.650, Y  +561.168, Z    +0.000, E1   -30.194, E3 +463872.873}
SPL {X  -165.650, Y  +565.528, Z    +0.000, E1   -30.192, E3 +463888.356}
SPL {X  -165.650, Y  +570.048, Z    +0.000, E1   -30.238, E3 +463903.787}
SPL {X  -165.650, Y  +573.110, Z    +0.000, E1   -30.057, E3 +463915.772}
SPL {X  -165.650, Y  +577.587, Z    +0.000, E1   -30.270, E3 +463930.211}
SPL {X  -165.650, Y  +581.190, Z    +0.000, E1   -30.107, E3 +463943.850}
SPL {X  -165.650, Y  +585.053, Z    +0.000, E1   -30.090, E3 +463957.720}
ENDSPLINE

SPLINE
SPL {X  -165.650, Y  +484.445, Z    +0.000, E1   +32.277, E3 +463975.125}
SPL {X  -165.650, Y  +481.524, Z    +0.000, E1   +31.089, E3 +463992.575}
SPL {X  -165.650, Y  +478.014, Z    +0.000, E1   +30.826, E3 +464006.183}
SPL {X  -165.650, Y  +474.473, Z    +0.000, E1   +30.943, E3 +464017.507}
SPL {X  -165.650, Y  +471.826, Z    +0.000, E1   +30.770, E3 +464027.691}
SPL {X  -165.650, Y  +467.753, Z    +0.000, E1   +30.878, E3 +464041.064}
SPL {X  -165.650, Y  +463.837, Z    +0.000, E1   +30.924, E3 +464053.998}
SPL {X  -165.650, Y  +461.106, Z    +0.000, E1   +30.916, E3 +464063.385}
SPL {X  -165.650, Y  +457.156, Z    +0.000, E1   +30.860, E3 +464077.461}
SPL {X  -165.650, Y  +453.156, Z    +0.000, E1   +30.934, E3 +464090.435}
SPL {X  -165.650, Y  +450.433, Z    +0.000, E1   +30.789, E3 +464100.791}
SPL {X  -165.650, Y  +447.097, Z    +0.000, E1   +30.843, E3 +464111.839}
SPL {X  -165.650, Y  +443.673, Z    +0.000, E1   +30.907, E3 +464123.147}
SPL {X  -165.650, Y  +439.486, Z    +0.000, E1   +30.857, E3 +464137.956}
SPL {X  -165.650, Y  +435.146, Z    +0.000, E1   +30.969, E3 +464151.876}
SPL {X  -165.650, Y  +432.765, Z    +0.000, E1   +30.831, E3 +464160.890}
SPL {X  -165.650, Y  +429.309, Z    +0.000, E1   +30.920, E3 +464172.231}
SPL {X  -165.650, Y  +424.918, Z    +0.000, E1   +30.862, E3 +464187.688}
SPL {X  -165.650, Y  +421.437, Z    +0.000, E1   +30.833, E3 +464199.656}
SPL {X  -165.650, Y  +417.366, Z    +0.000, E1   +30.879, E3 +464213.497}
SPL {X  -165.650, Y  +413.181, Z    +0.000, E1   +30.815, E3 +464228.094}
SPL {X  -165.650, Y  +408.547, Z    +0.000, E1   +30.964, E3 +464243.097}
SPL {X  -165.650, Y  +403.421, Z    +0.000, E1   +30.863, E3 +464261.315}
SPL {X  -165.650, Y  +399.681, Z    +0.000, E1   +30.933, E3 +464273.398}
SPL {X  -165.650, Y  +396.018, Z    +0.000, E1   +30.861, E3 +464286.708}
SPL {X  -165.650, Y  +391.522, Z    +0.000, E1   +30.837, E3 +464302.065}
SPL {X  -165.650, Y  +387.533, Z    +0.000, E1   +30.858, E3 +464315.691}
SPL {X  -165.650, Y  +383.627, Z    +0.000, E1   +30.885, E3 +464328.751}
SPL {X  -165.650, Y  +380.752, Z    +0.000, E1   +30.927, E3 +464338.265}
SPL {X  -165.648, Y  +377.739, Z    +0.000, E1   +30.835, E3 +464349.275}
SPL {X  -165.594, Y  +374.183, Z    +0.000, E1   +30.878, E3 +464361.111}
SPL {X  -165.429, Y  +369.945, Z    +0.000, E1   +30.850, E3 +464375.986}
SPL {X  -165.167, Y  +365.866, Z    +0.000, E1   +30.741, E3 +464390.519}
SPL {X  -164.892, Y  +362.671, Z    +0.000, E1   +30.830, E3 +464400.843}
SPL {X  -164.570, Y  +359.612, Z    +0.000, E1   +30.773, E3 +464411.656}
SPL {X  -164.287, Y  +357.291, Z    +0.000, E1   +30.513, E3 +464421.285}
SPL {X  -163.720, Y  +353.284, Z    +0.000, E1   +30.592, E3 +464434.732}
SPL {X  -162.976, Y  +348.856, Z    +0.000, E1   +30.757, E3 +464448.561}
SPL {X  -161.497, Y  +341.640, Z    +0.000, E1   +33.276, E3 +464455.838}
SPL {X  -152.976, Y  +314.952, Z    +0.000, E1   +38.607, E3 +464500.183}
SPL {X  -137.967, Y  +286.821, Z    +0.000, E1   +43.969, E3 +464543.404}
ENDSPLINE

SPLINE
SPL {X  -149.143, Y  +306.414, Z    +0.000, E1   +36.361, E3 +464594.536}
SPL {X  -164.268, Y  +357.145, Z    +0.000, E1   +15.880, E3 +464552.296}
SPL {X  -165.379, Y  +369.025, Z    +0.000, E1    +9.158, E3 +464556.967}
SPL {X  -165.612, Y  +374.969, Z    +0.000, E1    +5.630, E3 +464559.643}
SPL {X  -165.650, Y  +383.362, Z    +0.000, E1    +0.177, E3 +464544.261}
SPL {X  -165.650, Y  +383.923, Z    +0.000, E1    -0.215, E3 +464557.418}
SPL {X  -165.650, Y  +388.083, Z    +0.000, E1    -3.355, E3 +464556.282}
SPL {X  -165.650, Y  +393.983, Z    +0.000, E1    -8.501, E3 +464552.680}
SPL {X  -165.650, Y  +402.241, Z    +0.000, E1   -16.711, E3 +464547.192}
SPL {X  -165.650, Y  +416.345, Z    +0.000, E1   -29.511, E3 +464546.984}
SPL {X  -165.650, Y  +422.331, Z    +0.000, E1   -27.760, E3 +464572.483}
SPL {X  -165.650, Y  +441.276, Z    +0.000, E1   -37.343, E3 +464582.340}
SPL {X  -165.650, Y  +462.890, Z    +0.000, E1   -40.484, E3 +464616.423}
ENDSPLINE

SPLINE
SPL {X  -165.650, Y  +446.920, Z    +0.000, E1   -31.238, E3 +464628.749}
ENDSPLINE

SPLINE
SPL {X  -165.650, Y  +447.935, Z    +0.000, E1   -30.213, E3 +464639.037}
SPL {X  -165.650, Y  +451.020, Z    +0.000, E1   -30.224, E3 +464649.857}
SPL {X  -165.650, Y  +454.519, Z    +0.000, E1   -30.374, E3 +464661.039}
SPL {X  -165.650, Y  +457.429, Z    +0.000, E1   -30.029, E3 +464673.741}
SPL {X  -165.650, Y  +461.678, Z    +0.000, E1   -30.426, E3 +464685.866}
SPL {X  -165.650, Y  +463.853, Z    +0.000, E1   -30.103, E3 +464695.705}
SPL {X  -165.650, Y  +467.246, Z    +0.000, E1   -30.279, E3 +464706.436}
SPL {X  -165.650, Y  +469.780, Z    +0.000, E1   -30.237, E3 +464715.561}
SPL {X  -165.650, Y  +472.566, Z    +0.000, E1   -30.124, E3 +464726.219}
SPL {X  -165.650, Y  +475.265, Z    +0.000, E1   -30.034, E3 +464736.256}
SPL {X  -165.650, Y  +477.862, Z    +0.000, E1   -30.319, E3 +464743.448}
SPL {X  -165.650, Y  +481.042, Z    +0.000, E1   -30.192, E3 +464755.708}
SPL {X  -165.650, Y  +485.236, Z    +0.000, E1   -30.294, E3 +464769.563}
SPL {X  -165.650, Y  +488.041, Z    +0.000, E1   -30.253, E3 +464779.685}
SPL {X  -165.650, Y  +491.281, Z    +0.000, E1   -30.148, E3 +464791.823}
SPL {X  -165.650, Y  +495.051, Z    +0.000, E1   -30.213, E3 +464804.632}
SPL {X  -165.650, Y  +499.546, Z    +0.000, E1   -30.283, E3 +464820.074}
SPL {X  -165.650, Y  +503.544, Z    +0.000, E1   -30.247, E3 +464834.143}
SPL {X  -165.650, Y  +506.344, Z    +0.000, E1   -30.129, E3 +464844.811}
SPL {X  -165.650, Y  +509.866, Z    +0.000, E1   -30.236, E3 +464856.481}
SPL {X  -165.650, Y  +513.685, Z    +0.000, E1   -30.234, E3 +464869.977}
SPL {X  -165.650, Y  +517.919, Z    +0.000, E1   -30.227, E3 +464884.884}
SPL {X  -165.650, Y  +521.521, Z    +0.000, E1   -30.210, E3 +464897.559}
SPL {X  -165.650, Y  +525.344, Z    +0.000, E1   -30.269, E3 +464910.665}
SPL {X  -165.650, Y  +528.152, Z    +0.000, E1   -29.991, E3 +464922.306}
SPL {X  -165.650, Y  +531.783, Z    +0.000, E1   -30.416, E3 +464932.199}
SPL {X  -165.650, Y  +534.115, Z    +0.000, E1   -30.089, E3 +464942.581}
SPL {X  -165.650, Y  +537.522, Z    +0.000, E1   -30.251, E3 +464953.495}
SPL {X  -165.650, Y  +540.621, Z    +0.000, E1   -30.014, E3 +464966.056}
SPL {X  -165.650, Y  +544.944, Z    +0.000, E1   -30.447, E3 +464978.256}
SPL {X  -165.650, Y  +547.199, Z    +0.000, E1   -30.132, E3 +464988.229}
SPL {X  -165.650, Y  +550.512, Z    +0.000, E1   -30.197, E3 +464999.555}
SPL {X  -165.650, Y  +553.852, Z    +0.000, E1   -30.156, E3 +465011.496}
SPL {X  -165.650, Y  +557.277, Z    +0.000, E1   -30.150, E3 +465023.670}
SPL {X  -165.650, Y  +561.168, Z    +0.000, E1   -30.194, E3 +465037.052}
SPL {X  -165.650, Y  +564.449, Z    +0.000, E1   -30.167, E3 +465048.735}
SPL {X  -165.650, Y  +566.935, Z    +0.000, E1   -30.135, E3 +465057.641}
SPL {X  -165.650, Y  +570.048, Z    +0.000, E1   -30.238, E3 +465067.966}
SPL {X  -165.650, Y  +573.110, Z    +0.000, E1   -30.057, E3 +465079.951}
SPL {X  -165.650, Y  +577.587, Z    +0.000, E1   -30.270, E3 +465094.390}
SPL {X  -165.650, Y  +581.190, Z    +0.000, E1   -30.107, E3 +465108.029}
SPL {X  -165.650, Y  +585.053, Z    +0.000, E1   -30.090, E3 +465121.899}
ENDSPLINE

SPLINE
SPL {X  -165.650, Y  +484.445, Z    +0.000, E1   +32.277, E3 +465139.304}
SPL {X  -165.650, Y  +481.524, Z    +0.000, E1   +31.089, E3 +465156.754}
SPL {X  -165.650, Y  +478.014, Z    +0.000, E1   +30.826, E3 +465170.362}
SPL {X  -165.650, Y  +474.473, Z    +0.000, E1   +30.943, E3 +465181.686}
SPL {X  -165.650, Y  +471.826, Z    +0.000, E1   +30.770, E3 +465191.870}
SPL {X  -165.650, Y  +467.753, Z    +0.000, E1   +30.878, E3 +465205.243}
SPL {X  -165.650, Y  +463.837, Z    +0.000, E1   +30.924, E3 +465218.177}
SPL {X  -165.650, Y  +461.106, Z    +0.000, E1   +30.916, E3 +465227.564}
SPL {X  -165.650, Y  +458.435, Z    +0.000, E1   +30.759, E3 +465237.772}
SPL {X  -165.650, Y  +454.220, Z    +0.000, E1   +30.954, E3 +465251.005}
SPL {X  -165.650, Y  +450.433, Z    +0.000, E1   +30.789, E3 +465264.970}
SPL {X  -165.650, Y  +447.097, Z    +0.000, E1   +30.843, E3 +465276.018}
SPL {X  -165.650, Y  +443.673, Z    +0.000, E1   +30.907, E3 +465287.326}
SPL {X  -165.650, Y  +440.976, Z    +0.000, E1   +30.719, E3 +465297.783}
SPL {X  -165.650, Y  +436.324, Z    +0.000, E1   +30.994, E3 +465312.069}
SPL {X  -165.650, Y  +432.765, Z    +0.000, E1   +30.831, E3 +465325.069}
SPL {X  -165.650, Y  +429.309, Z    +0.000, E1   +30.920, E3 +465336.410}
SPL {X  -165.650, Y  +424.918, Z    +0.000, E1   +30.862, E3 +465351.867}
SPL {X  -165.650, Y  +421.437, Z    +0.000, E1   +30.833, E3 +465363.835}
SPL {X  -165.650, Y  +418.489, Z    +0.000, E1   +30.835, E3 +465373.952}
SPL {X  -165.650, Y  +414.127, Z    +0.000, E1   +30.869, E3 +465388.861}
SPL {X  -165.650, Y  +408.547, Z    +0.000, E1   +30.964, E3 +465407.276}
SPL {X  -165.650, Y  +405.433, Z    +0.000, E1   +30.730, E3 +465419.253}
SPL {X  -165.650, Y  +402.516, Z    +0.000, E1   +30.874, E3 +465428.376}
SPL {X  -165.650, Y  +398.147, Z    +0.000, E1   +30.902, E3 +465443.255}
SPL {X  -165.650, Y  +394.694, Z    +0.000, E1   +30.805, E3 +465455.563}
SPL {X  -165.650, Y  +391.522, Z    +0.000, E1   +30.837, E3 +465466.244}
SPL {X  -165.650, Y  +387.533, Z    +0.000, E1   +30.858, E3 +465479.870}
SPL {X  -165.650, Y  +383.627, Z    +0.000, E1   +30.885, E3 +465492.930}
SPL {X  -165.650, Y  +379.886, Z    +0.000, E1   +30.887, E3 +465505.819}
SPL {X  -165.614, Y  +375.058, Z    +0.000, E1   +30.905, E3 +465522.272}
SPL {X  -165.492, Y  +371.263, Z    +0.000, E1   +30.913, E3 +465534.986}
SPL {X  -165.379, Y  +369.027, Z    +0.000, E1   +30.727, E3 +465543.924}
SPL {X  -165.167, Y  +365.866, Z    +0.000, E1   +30.741, E3 +465554.698}
SPL {X  -164.892, Y  +362.671, Z    +0.000, E1   +30.830, E3 +465565.022}
SPL {X  -164.570, Y  +359.612, Z    +0.000, E1   +30.773, E3 +465575.835}
SPL {X  -164.104, Y  +355.923, Z    +0.000, E1   +30.626, E3 +465589.551}
SPL {X  -163.573, Y  +352.353, Z    +0.000, E1   +30.451, E3 +465602.816}
SPL {X  -162.476, Y  +346.230, Z    +0.000, E1   +31.677, E3 +465615.397}
SPL {X  -152.976, Y  +314.952, Z    +0.000, E1   +38.607, E3 +465664.362}
SPL {X  -137.967, Y  +286.821, Z    +0.000, E1   +43.969, E3 +465707.583}
ENDSPLINE

SPLINE
SPL {X  -149.143, Y  +306.414, Z    +0.000, E1   +36.361, E3 +465758.716}
SPL {X  -164.268, Y  +357.145, Z    +0.000, E1   +15.880, E3 +465716.475}
SPL {X  -165.510, Y  +371.680, Z    +0.000, E1    +7.684, E3 +465719.477}
SPL {X  -165.628, Y  +375.818, Z    +0.000, E1    +5.016, E3 +465727.407}
SPL {X  -165.650, Y  +383.362, Z    +0.000, E1    +0.177, E3 +465708.440}
SPL {X  -165.650, Y  +383.923, Z    +0.000, E1    -0.215, E3 +465721.598}
SPL {X  -165.650, Y  +388.083, Z    +0.000, E1    -3.355, E3 +465720.461}
SPL {X  -165.650, Y  +393.983, Z    +0.000, E1    -8.501, E3 +465716.859}
SPL {X  -165.650, Y  +402.241, Z    +0.000, E1   -16.711, E3 +465711.371}
SPL {X  -165.650, Y  +416.345, Z    +0.000, E1   -29.511, E3 +465711.163}
SPL {X  -165.650, Y  +422.331, Z    +0.000, E1   -27.760, E3 +465736.662}
SPL {X  -165.650, Y  +441.276, Z    +0.000, E1   -37.343, E3 +465746.519}
SPL {X  -165.650, Y  +462.890, Z    +0.000, E1   -40.484, E3 +465780.602}
ENDSPLINE

SPLINE
SPL {X  -165.650, Y  +446.920, Z    +0.000, E1   -31.238, E3 +465792.928}
ENDSPLINE

SPLINE
SPL {X  -165.650, Y  +447.935, Z    +0.000, E1   -30.213, E3 +465803.216}
SPL {X  -165.650, Y  +451.020, Z    +0.000, E1   -30.224, E3 +465814.036}
SPL {X  -165.650, Y  +454.519, Z    +0.000, E1   -30.374, E3 +465825.219}
SPL {X  -165.650, Y  +456.542, Z    +0.000, E1   -29.986, E3 +465834.963}
SPL {X  -165.650, Y  +460.618, Z    +0.000, E1   -30.298, E3 +465847.284}
SPL {X  -165.650, Y  +463.853, Z    +0.000, E1   -30.103, E3 +465859.885}
SPL {X  -165.650, Y  +468.397, Z    +0.000, E1   -30.302, E3 +465874.688}
SPL {X  -165.650, Y  +472.566, Z    +0.000, E1   -30.124, E3 +465890.398}
SPL {X  -165.650, Y  +475.265, Z    +0.000, E1   -30.034, E3 +465900.435}
SPL {X  -165.650, Y  +477.862, Z    +0.000, E1   -30.319, E3 +465907.627}
SPL {X  -165.650, Y  +481.042, Z    +0.000, E1   -30.192, E3 +465919.887}
SPL {X  -165.650, Y  +485.236, Z    +0.000, E1   -30.294, E3 +465933.743}
SPL {X  -165.650, Y  +488.041, Z    +0.000, E1   -30.253, E3 +465943.864}
SPL {X  -165.650, Y  +491.281, Z    +0.000, E1   -30.148, E3 +465956.002}
SPL {X  -165.650, Y  +495.051, Z    +0.000, E1   -30.213, E3 +465968.811}
SPL {X  -165.650, Y  +499.546, Z    +0.000, E1   -30.283, E3 +465984.253}
SPL {X  -165.650, Y  +503.544, Z    +0.000, E1   -30.247, E3 +465998.322}
SPL {X  -165.650, Y  +506.344, Z    +0.000, E1   -30.129, E3 +466008.991}
SPL {X  -165.650, Y  +510.660, Z    +0.000, E1   -30.223, E3 +466023.694}
SPL {X  -165.650, Y  +514.670, Z    +0.000, E1   -30.278, E3 +466037.204}
SPL {X  -165.650, Y  +517.919, Z    +0.000, E1   -30.227, E3 +466049.063}
SPL {X  -165.650, Y  +521.521, Z    +0.000, E1   -30.210, E3 +466061.738}
SPL {X  -165.650, Y  +525.344, Z    +0.000, E1   -30.269, E3 +466074.844}
SPL {X  -165.650, Y  +528.152, Z    +0.000, E1   -29.991, E3 +466086.485}
SPL {X  -165.650, Y  +531.783, Z    +0.000, E1   -30.416, E3 +466096.378}
SPL {X  -165.650, Y  +534.115, Z    +0.000, E1   -30.089, E3 +466106.760}
SPL {X  -165.650, Y  +537.522, Z    +0.000, E1   -30.251, E3 +466117.674}
SPL {X  -165.650, Y  +540.621, Z    +0.000, E1   -30.014, E3 +466130.235}
SPL {X  -165.650, Y  +544.944, Z    +0.000, E1   -30.447, E3 +466142.435}
SPL {X  -165.650, Y  +547.199, Z    +0.000, E1   -30.132, E3 +466152.408}
SPL {X  -165.650, Y  +550.512, Z    +0.000, E1   -30.197, E3 +466163.734}
SPL {X  -165.650, Y  +553.852, Z    +0.000, E1   -30.156, E3 +466175.675}
SPL {X  -165.650, Y  +557.277, Z    +0.000, E1   -30.150, E3 +466187.849}
SPL {X  -165.650, Y  +561.168, Z    +0.000, E1   -30.194, E3 +466201.231}
SPL {X  -165.650, Y  +565.528, Z    +0.000, E1   -30.192, E3 +466216.714}
SPL {X  -165.650, Y  +570.048, Z    +0.000, E1   -30.238, E3 +466232.145}
SPL {X  -165.650, Y  +573.110, Z    +0.000, E1   -30.057, E3 +466244.130}
SPL {X  -165.650, Y  +577.587, Z    +0.000, E1   -30.270, E3 +466258.569}
SPL {X  -165.650, Y  +581.190, Z    +0.000, E1   -30.107, E3 +466272.208}
SPL {X  -165.650, Y  +585.053, Z    +0.000, E1   -30.090, E3 +466286.078}
ENDSPLINE

SPLINE
SPL {X  -165.650, Y  +484.445, Z    +0.000, E1   +32.277, E3 +466303.483}
SPL {X  -165.650, Y  +481.524, Z    +0.000, E1   +31.089, E3 +466320.933}
SPL {X  -165.650, Y  +478.014, Z    +0.000, E1   +30.826, E3 +466334.541}
SPL {X  -165.650, Y  +474.473, Z    +0.000, E1   +30.943, E3 +466345.865}
SPL {X  -165.650, Y  +470.376, Z    +0.000, E1   +30.888, E3 +466360.395}
SPL {X  -165.650, Y  +465.146, Z    +0.000, E1   +30.883, E3 +466378.325}
SPL {X  -165.650, Y  +461.106, Z    +0.000, E1   +30.916, E3 +466391.743}
SPL {X  -165.650, Y  +458.435, Z    +0.000, E1   +30.759, E3 +466401.951}
SPL {X  -165.650, Y  +454.220, Z    +0.000, E1   +30.954, E3 +466415.184}
SPL {X  -165.650, Y  +450.433, Z    +0.000, E1   +30.789, E3 +466429.149}
SPL {X  -165.650, Y  +447.097, Z    +0.000, E1   +30.843, E3 +466440.198}
SPL {X  -165.650, Y  +443.673, Z    +0.000, E1   +30.907, E3 +466451.505}
SPL {X  -165.650, Y  +440.976, Z    +0.000, E1   +30.719, E3 +466461.962}
SPL {X  -165.650, Y  +436.324, Z    +0.000, E1   +30.994, E3 +466476.248}
SPL {X  -165.650, Y  +432.765, Z    +0.000, E1   +30.831, E3 +466489.248}
SPL {X  -165.650, Y  +429.309, Z    +0.000, E1   +30.920, E3 +466500.589}
SPL {X  -165.650, Y  +424.918, Z    +0.000, E1   +30.862, E3 +466516.046}
SPL {X  -165.650, Y  +421.437, Z    +0.000, E1   +30.833, E3 +466528.015}
SPL {X  -165.650, Y  +417.366, Z    +0.000, E1   +30.879, E3 +466541.855}
SPL {X  -165.650, Y  +412.139, Z    +0.000, E1   +30.870, E3 +466559.805}
SPL {X  -165.650, Y  +406.834, Z    +0.000, E1   +30.919, E3 +466577.633}
SPL {X  -165.650, Y  +402.516, Z    +0.000, E1   +30.874, E3 +466592.555}
SPL {X  -165.650, Y  +398.147, Z    +0.000, E1   +30.902, E3 +466607.434}
SPL {X  -165.650, Y  +394.694, Z    +0.000, E1   +30.805, E3 +466619.742}
SPL {X  -165.650, Y  +391.522, Z    +0.000, E1   +30.837, E3 +466630.423}
SPL {X  -165.650, Y  +387.533, Z    +0.000, E1   +30.858, E3 +466644.049}
SPL {X  -165.650, Y  +383.627, Z    +0.000, E1   +30.885, E3 +466657.109}
SPL {X  -165.650, Y  +380.752, Z    +0.000, E1   +30.927, E3 +466666.623}
SPL {X  -165.648, Y  +377.739, Z    +0.000, E1   +30.835, E3 +466677.633}
SPL {X  -165.594, Y  +374.183, Z    +0.000, E1   +30.878, E3 +466689.470}
SPL {X  -165.492, Y  +371.263, Z    +0.000, E1   +30.913, E3 +466699.165}
SPL {X  -165.379, Y  +369.027, Z    +0.000, E1   +30.727, E3 +466708.103}
SPL {X  -165.167, Y  +365.866, Z    +0.000, E1   +30.741, E3 +466718.877}
SPL {X  -164.892, Y  +362.671, Z    +0.000, E1   +30.830, E3 +466729.201}
SPL {X  -164.570, Y  +359.612, Z    +0.000, E1   +30.773, E3 +466740.014}
SPL {X  -164.104, Y  +355.923, Z    +0.000, E1   +30.626, E3 +466753.730}
SPL {X  -163.573, Y  +352.353, Z    +0.000, E1   +30.451, E3 +466766.995}
SPL {X  -162.476, Y  +346.230, Z    +0.000, E1   +31.677, E3 +466779.576}
SPL {X  -152.976, Y  +314.952, Z    +0.000, E1   +38.607, E3 +466828.541}
SPL {X  -137.967, Y  +286.821, Z    +0.000, E1   +43.969, E3 +466871.762}
ENDSPLINE

SPLINE
SPL {X  -153.316, Y  +315.777, Z    +0.000, E1   +33.140, E3 +466914.390}
SPL {X  -164.446, Y  +358.564, Z    +0.000, E1   +15.149, E3 +466879.601}
SPL {X  -165.379, Y  +369.025, Z    +0.000, E1    +9.158, E3 +466885.325}
SPL {X  -165.612, Y  +374.969, Z    +0.000, E1    +5.630, E3 +466888.001}
SPL {X  -165.650, Y  +383.362, Z    +0.000, E1    +0.177, E3 +466872.619}
SPL {X  -165.650, Y  +383.923, Z    +0.000, E1    -0.215, E3 +466885.777}
SPL {X  -165.650, Y  +388.083, Z    +0.000, E1    -3.355, E3 +466884.640}
SPL {X  -165.650, Y  +393.983, Z    +0.000, E1    -8.501, E3 +466881.038}
SPL {X  -165.650, Y  +402.241, Z    +0.000, E1   -16.711, E3 +466875.550}
SPL {X  -165.650, Y  +416.345, Z    +0.000, E1   -29.511, E3 +466875.342}
SPL {X  -165.650, Y  +422.331, Z    +0.000, E1   -27.760, E3 +466900.841}
SPL {X  -165.650, Y  +441.276, Z    +0.000, E1   -37.343, E3 +466910.698}
SPL {X  -165.650, Y  +462.890, Z    +0.000, E1   -40.484, E3 +466944.781}
ENDSPLINE

SPLINE
SPL {X  -165.650, Y  +446.920, Z    +0.000, E1   -31.238, E3 +466957.107}
ENDSPLINE

SPLINE
SPL {X  -165.650, Y  +447.935, Z    +0.000, E1   -30.213, E3 +466967.395}
SPL {X  -165.650, Y  +451.020, Z    +0.000, E1   -30.224, E3 +466978.215}
SPL {X  -165.650, Y  +454.519, Z    +0.000, E1   -30.374, E3 +466989.398}
SPL {X  -165.650, Y  +456.542, Z    +0.000, E1   -29.986, E3 +466999.142}
SPL {X  -165.650, Y  +460.618, Z    +0.000, E1   -30.298, E3 +467011.463}
SPL {X  -165.650, Y  +463.853, Z    +0.000, E1   -30.103, E3 +467024.064}
SPL {X  -165.650, Y  +467.246, Z    +0.000, E1   -30.279, E3 +467034.794}
SPL {X  -165.650, Y  +469.780, Z    +0.000, E1   -30.237, E3 +467043.919}
SPL {X  -165.650, Y  +472.566, Z    +0.000, E1   -30.124, E3 +467054.577}
SPL {X  -165.650, Y  +476.540, Z    +0.000, E1   -30.193, E3 +467068.121}
SPL {X  -165.650, Y  +480.320, Z    +0.000, E1   -30.163, E3 +467081.599}
SPL {X  -165.650, Y  +484.477, Z    +0.000, E1   -30.274, E3 +467095.488}
SPL {X  -165.650, Y  +488.041, Z    +0.000, E1   -30.253, E3 +467108.043}
SPL {X  -165.650, Y  +491.281, Z    +0.000, E1   -30.148, E3 +467120.181}
SPL {X  -165.650, Y  +495.051, Z    +0.000, E1   -30.213, E3 +467132.990}
SPL {X  -165.650, Y  +498.418, Z    +0.000, E1   -30.282, E3 +467144.283}
SPL {X  -165.650, Y  +500.833, Z    +0.000, E1   -30.191, E3 +467153.332}
SPL {X  -165.650, Y  +504.246, Z    +0.000, E1   -30.231, E3 +467165.198}
SPL {X  -165.650, Y  +507.017, Z    +0.000, E1   -30.108, E3 +467175.606}
SPL {X  -165.650, Y  +510.660, Z    +0.000, E1   -30.223, E3 +467187.873}
SPL {X  -165.650, Y  +515.918, Z    +0.000, E1   -30.316, E3 +467205.681}
SPL {X  -165.650, Y  +520.621, Z    +0.000, E1   -30.198, E3 +467222.967}
SPL {X  -165.650, Y  +525.344, Z    +0.000, E1   -30.269, E3 +467239.023}
SPL {X  -165.650, Y  +528.152, Z    +0.000, E1   -29.991, E3 +467250.664}
SPL {X  -165.650, Y  +531.783, Z    +0.000, E1   -30.416, E3 +467260.557}
SPL {X  -165.650, Y  +534.115, Z    +0.000, E1   -30.089, E3 +467270.939}
SPL {X  -165.650, Y  +538.363, Z    +0.000, E1   -30.232, E3 +467285.109}
SPL {X  -165.650, Y  +543.650, Z    +0.000, E1   -30.281, E3 +467303.329}
SPL {X  -165.650, Y  +547.199, Z    +0.000, E1   -30.132, E3 +467316.588}
SPL {X  -165.650, Y  +550.512, Z    +0.000, E1   -30.197, E3 +467327.913}
SPL {X  -165.650, Y  +554.908, Z    +0.000, E1   -30.180, E3 +467343.575}
SPL {X  -165.650, Y  +560.243, Z    +0.000, E1   -30.214, E3 +467362.200}
SPL {X  -165.650, Y  +565.528, Z    +0.000, E1   -30.192, E3 +467380.893}
SPL {X  -165.650, Y  +570.048, Z    +0.000, E1   -30.238, E3 +467396.324}
SPL {X  -165.650, Y  +573.110, Z    +0.000, E1   -30.057, E3 +467408.309}
SPL {X  -165.650, Y  +577.587, Z    +0.000, E1   -30.270, E3 +467422.748}
SPL {X  -165.650, Y  +581.190, Z    +0.000, E1   -30.107, E3 +467436.387}
SPL {X  -165.650, Y  +585.053, Z    +0.000, E1   -30.090, E3 +467450.257}
ENDSPLINE

